# B&R Automation Studio project 8238 (part 20)

#### _actReqScheduleDFII.st
```iecst
(********************************************************************
 * COPYRIGHT -- Herbert Kannegiesser GmbH
 ********************************************************************
 * Program: hlDFII
 * File: _actReqScheduleDFII.st
 * Author: hunholz
 * Created: June 20, 2012
 ********************************************************************
 * Implementation of program hlDFII
 ********************************************************************)

(* Process Requests for DFII *)
ACTION _actReqScheduleDFII:

	// Der Scheduler wird nur ausgeführt, wenn kein SQL-Commando bearbeitet wird

	IF _eCmdDFIIStep = eCMD_SQLREQ_IDLE THEN

		CASE _wScheduleStep OF

			_HLDFII_SCHEDSTEP_GETTIME:

				// Uhrzeit holen
				IF _bEventGetTime = _HLDFII_REQ_START THEN
					// Auftrag starten
					_eCmdDFIIStep := eCMD_SQLREQ_WRITE_GETTIME;
					_bEventGetTime := _HLDFII_REQ_RUN;
				END_IF

			_HLDFII_SCHEDSTEP_REGMACHINE:

				// Maschine registrieren
				IF _bEventRegMach = _HLDFII_REQ_START AND brwcscmp(ADR(IFmnParam.Out.utfMachineNumber),ADR(MNPARAM_INVALID_MACHINENO)) <> 0 THEN
					// Auftrag starten
					_eCmdDFIIStep := eCMD_SQLREQ_WRITE_REGMACH;
					_bEventRegMach := _HLDFII_REQ_RUN;
				END_IF

			_HLDFII_SCHEDSTEP_PROGBYCAT:

				// Programmnummer anhand der Kategorie ermitteln
				IF _xWaitReqProgByCatIsZero THEN

					IF IFhlDFII.In.ReqProgByCat.wRequest = 0 THEN

						_xWaitReqProgByCatIsZero := FALSE;
						IFhlDFII.Out.RespProgByCat.wResponse := 0;

					END_IF

				ELSE

					// Prüfen ob eine Programmnummer gelesen werden soll
					IF IFhlDFII.In.ReqProgByCat.wRequest = 1 OR IFhlDFII.In.ReqProgByCat.wRequest = 2 THEN

						IF IFhlDFII.Out.xConnected THEN

							_xWaitReqProgByCatIsZero := TRUE;
							// Auftrag starten
							_eCmdDFIIStep := eCMD_SQLREQ_GET_PROG_BY_CAT;
							IFhlDFII.Out.RespProgByCat.wResponse := ERR_FUB_BUSY;

						ELSE

							_xWaitReqProgByCatIsZero := TRUE;
							IFhlDFII.Out.RespProgByCat.wResponse := HLDFII_STAT_NO_CONNECTION;

						END_IF

					END_IF

				END_IF

			_HLDFII_SCHEDSTEP_MSGEVENT:

				// Meldungden senden
				IF _xWaitReqMsgEvtIsZero THEN

					IF IFhlDFII.In.ReqMsgEvt.wRequest = 0 THEN
						_xWaitReqMsgEvtIsZero := FALSE;
						IFhlDFII.Out.RespMsgEvt.wResponse := 0;
					END_IF

				ELSE

					IF IFhlDFII.Out.xConnected THEN

						// Prüfen ob Meldungsevents geschrieben werden sollen
						IF IFhlDFII.In.ReqMsgEvt.wRequest = 1 THEN

							_xWaitReqMsgEvtIsZero := TRUE;

							IF IFhlDFII.In.ReqMsgEvt.bCntLines > 0 THEN
								_eCmdDFIIStep := eCMD_SQLREQ_WRITE_MSG;
								IFhlDFII.Out.RespMsgEvt.wResponse := ERR_FUB_BUSY;
							ELSE
								IFhlDFII.Out.RespMsgEvt.wResponse := IFhlDFII.In.ReqMsgEvt.wRequest;
							END_IF

						END_IF

					ELSE

						_xWaitReqMsgEvtIsZero := TRUE;
						IFhlDFII.Out.RespMsgEvt.wResponse := HLDFII_STAT_NO_CONNECTION;

					END_IF

				END_IF

			_HLDFII_SCHEDSTEP_CNTBATCH:

				// Postendaten senden
				IF _xWaitReqCntBatchIsZero THEN

					IF IFhlDFII.In.ReqCntBatchEvt.wRequest = 0 THEN

						_xWaitReqCntBatchIsZero := FALSE;
						IFhlDFII.Out.RespCntBatchEvt.wResponse := 0;

					END_IF

				ELSE

					IF IFhlDFII.Out.xConnected THEN

						// Prüfen ob Zähler-Posten-Events geschrieben werden sollen
						IF IFhlDFII.In.ReqCntBatchEvt.wRequest = 1 THEN

							_xWaitReqCntBatchIsZero := TRUE;

							IF IFhlDFII.In.ReqCntBatchEvt.bCntLines > 0 THEN
								_eCmdDFIIStep := eCMD_SQLREQ_WRITE_CNTBATCHEVT;
								IFhlDFII.Out.RespCntBatchEvt.wResponse := ERR_FUB_BUSY;
							ELSE
								IFhlDFII.Out.RespCntBatchEvt.wResponse  := IFhlDFII.In.ReqCntBatchEvt.wRequest;
							END_IF
						END_IF

					ELSE

						_xWaitReqCntBatchIsZero := TRUE;
						IFhlDFII.Out.RespCntBatchEvt.wResponse := HLDFII_STAT_NO_CONNECTION;

					END_IF

				END_IF

			// Zähler senden
			_HLDFII_SCHEDSTEP_CNTCNT:

				IF _xWaitReqCntCntIsZero THEN

					IF IFhlDFII.In.ReqCntCntEvt.wRequest = 0 THEN

						_xWaitReqCntCntIsZero := FALSE;
						IFhlDFII.Out.RespCntCntEvt.wResponse := 0;

					END_IF

				ELSE

					IF IFhlDFII.Out.xConnected THEN

						// Prüfen ob Zähler-Zähler-Events geschrieben werden sollen
						IF IFhlDFII.In.ReqCntCntEvt.wRequest = 1 THEN

							_xWaitReqCntCntIsZero := TRUE;

							IF IFhlDFII.In.ReqCntCntEvt.bCntLines > 0 THEN
								_eCmdDFIIStep := eCMD_SQLREQ_WRITE_CNTCNTEVT;
								IFhlDFII.Out.RespCntCntEvt.wResponse := ERR_FUB_BUSY;
							ELSE
								IFhlDFII.Out.RespCntCntEvt.wResponse  := IFhlDFII.In.ReqCntCntEvt.wRequest;
							END_IF
						END_IF

					ELSE

						_xWaitReqCntCntIsZero := TRUE;
						IFhlDFII.Out.RespCntCntEvt.wResponse := HLDFII_STAT_NO_CONNECTION;

					END_IF

				END_IF

			// Zeiten senden
			_HLDFII_SCHEDSTEP_CNTTIME:

				IF _xWaitReqCntTimIsZero THEN

					IF IFhlDFII.In.ReqCntTimEvt.wRequest = 0 THEN

						_xWaitReqCntTimIsZero := FALSE;
						IFhlDFII.Out.RespCntTimEvt.wResponse := 0;

					END_IF

				ELSE

					IF IFhlDFII.Out.xConnected THEN

						// Prüfen ob Zähler-Zeit-Events geschrieben werden sollen
						IF IFhlDFII.In.ReqCntTimEvt.wRequest = 1 THEN

							_xWaitReqCntTimIsZero := TRUE;

							IF IFhlDFII.In.ReqCntTimEvt.bCntLines > 0 THEN
								_eCmdDFIIStep := eCMD_SQLREQ_WRITE_CNTTIMEVT;
								IFhlDFII.Out.RespCntTimEvt.wResponse := ERR_FUB_BUSY;
							ELSE
								IFhlDFII.Out.RespCntTimEvt.wResponse  := IFhlDFII.In.ReqCntTimEvt.wRequest;
							END_IF
						END_IF

					ELSE

						_xWaitReqCntTimIsZero := TRUE;
						IFhlDFII.Out.RespCntTimEvt.wResponse := HLDFII_STAT_NO_CONNECTION;

					END_IF

				END_IF

			// Dosierungen senden
			_HLDFII_SCHEDSTEP_CNTDOS:

				IF _xWaitReqCntDosIsZero THEN

					IF IFhlDFII.In.ReqCntDosEvt.wRequest = 0 THEN

						_xWaitReqCntDosIsZero := FALSE;
						IFhlDFII.Out.RespCntDosEvt.wResponse := 0;

					END_IF

				ELSE

					IF IFhlDFII.Out.xConnected THEN

						// Prüfen ob Zähler-Dosier-Events geschrieben werden sollen
						IF IFhlDFII.In.ReqCntDosEvt.wRequest = 1 THEN

							_xWaitReqCntDosIsZero := TRUE;

							IF IFhlDFII.In.ReqCntDosEvt.bCntLines > 0 THEN
								_eCmdDFIIStep := eCMD_SQLREQ_WRITE_CNTDOSEVT;
								IFhlDFII.Out.RespCntDosEvt.wResponse := ERR_FUB_BUSY;
							ELSE
								IFhlDFII.Out.RespCntDosEvt.wResponse  := IFhlDFII.In.ReqCntDosEvt.wRequest;
							END_IF

						END_IF

					ELSE

						_xWaitReqCntDosIsZero := TRUE;
						IFhlDFII.Out.RespCntDosEvt.wResponse := HLDFII_STAT_NO_CONNECTION;

					END_IF

				END_IF

		END_CASE

	END_IF

END_ACTION
```

#### _actProcCmdTrack.st
```iecst
(********************************************************************
 * COPYRIGHT -- Herbert Kannegiesser GmbH
 ********************************************************************
 * Program: hlDFII
 * File: _actProcCmdTrack.st
 * Author: hunholz
 * Created: June 20, 2012
 ********************************************************************
 * Implementation of program hlDFII
 ********************************************************************)

(* Process Commands for DFII *)
ACTION _actProcCmdTrack:

	_TONRefreshTrack(IN := NOT _TONRefreshTrack.Q, PT := T#1s);

	CASE _eCmdTrackStep OF

		//*****************************************************
		// Im Idle Zustand werden laufend die Auftrage gescannt
		//*****************************************************
		eCMD_SQLREQ_IDLE:

			// Zuerst wird die Zeit vom Server geholt
			IF _bEventGetTrackTime <> _HLDFII_REQ_FINISHED THEN

				_wScheduleTrackStep := _HLDFII_SCHEDSTEP_T_GETTIME;

				// Dann wird zyklisch geschaut, ob Anforderungen anliegen
			ELSE

				IF _TONRefreshTrack.Q THEN

					_wScheduleTrackStepHelp := (_wScheduleTrackStepHelp + 1) MOD (_HLDFII_SCHEDSTEP_T_MAX);

					_wScheduleTrackStep := _wScheduleTrackStepHelp + 1;

				END_IF

			END_IF

		//*****************************************************
		// Uhrzeit vom DB-Server holen
		//*****************************************************
		eCMD_SQLREQ_WRITE_GETTIME:

			IF _eTrackStep = eSQLREQ_STEP_WAITFORCOMMAND THEN

				_eTrackStep := eSQLREQ_STEP_GETTIME;
				_eCmdTrackStep := eCMD_SQLREQ_WRITE_GETTIME_w;

			ELSIF _eTrackStep = eSQLREQ_STEP_ERROR THEN

				_bEventGetTrackTime := _HLDFII_REQ_FAULT;
				_eCmdTrackStep := eCMD_SQLREQ_IDLE;

			END_IF

		eCMD_SQLREQ_WRITE_GETTIME_w:

			IF _eTrackStep = eSQLREQ_STEP_WAITFORCOMMAND THEN

				_bEventGetTrackTime := _HLDFII_REQ_FINISHED;
				_eCmdTrackStep := eCMD_SQLREQ_IDLE;

			ELSIF _eTrackStep = eSQLREQ_STEP_ERROR THEN

				_bEventGetTrackTime := _HLDFII_REQ_FAULT;
				_eCmdTrackStep := eCMD_SQLREQ_IDLE;

			END_IF

		//***************************************
		// Batchdaten in Location-Table eintragen
		//***************************************
		eCMD_SQLREQ_WRITE_UPDLOC:

			IF _eTrackStep = eSQLREQ_STEP_WAITFORCOMMAND THEN

				_wIdxWriteUpdateLocation := 1;
				_eTrackStep := eSQLREQ_STEP_WRUPDLOC;
				_eCmdTrackStep := eCMD_SQLREQ_WRITE_UPDLOC_w;

			ELSIF _eTrackStep = eSQLREQ_STEP_ERROR THEN

				_xUpdateLocationFinished := TRUE;
				_eCmdTrackStep := eCMD_SQLREQ_IDLE;

			END_IF

		eCMD_SQLREQ_WRITE_UPDLOC_w:

			IF _eTrackStep = eSQLREQ_STEP_WAITFORCOMMAND THEN

				_xUpdateLocationFinished := TRUE;
				_eCmdTrackStep := eCMD_SQLREQ_IDLE;

			ELSIF _eTrackStep = eSQLREQ_STEP_ERROR THEN

				_xUpdateLocationFinished := TRUE;
				_eCmdTrackStep := eCMD_SQLREQ_IDLE;

			END_IF

		//***************************************
		// Maschinenstatus eintragen
		//***************************************
		eCMD_SQLREQ_WRITE_UPDSTATE:

			IF _eTrackStep = eSQLREQ_STEP_WAITFORCOMMAND THEN

				_wIdxWriteUpdateStatus := 1;
				_eTrackStep := eSQLREQ_STEP_WRUPDSTATE;
				_eCmdTrackStep := eCMD_SQLREQ_WRITE_UPDSTATE_w;

			ELSIF _eTrackStep = eSQLREQ_STEP_ERROR THEN

				_xUpdateStatusFinished := TRUE;
				_eCmdTrackStep := eCMD_SQLREQ_IDLE;

			END_IF

		eCMD_SQLREQ_WRITE_UPDSTATE_w:

			IF _eTrackStep = eSQLREQ_STEP_WAITFORCOMMAND THEN

				_xUpdateStatusFinished := TRUE;
				_eCmdTrackStep := eCMD_SQLREQ_IDLE;

			ELSIF _eTrackStep = eSQLREQ_STEP_ERROR THEN

				_xUpdateStatusFinished := TRUE;
				_eCmdTrackStep := eCMD_SQLREQ_IDLE;

			END_IF

	END_CASE

END_ACTION
```

#### _actProcCmdDFII.st
```iecst
(********************************************************************
 * COPYRIGHT -- Herbert Kannegiesser GmbH
 ********************************************************************
 * Program: hlDFII
 * File: _actProcCmdDFII.st
 * Author: hunholz
 * Created: June 20, 2012
 ********************************************************************
 * Implementation of program hlDFII
 ********************************************************************)

(* Process Commands for DFII *)
ACTION _actProcCmdDFII:

	CASE _eCmdDFIIStep OF

		//*****************************************************
		// Im Idle Zustand werden laufend die Auftrage gescannt
		//*****************************************************
		eCMD_SQLREQ_IDLE:

			// Zuerst wird die Zeit vom Server geholt
			IF _bEventGetTime <> _HLDFII_REQ_FINISHED THEN

				_wScheduleStep := _HLDFII_SCHEDSTEP_GETTIME;

				// Die Maschine wird auf jeden Fall registriert
			ELSIF _bEventRegMach <> _HLDFII_REQ_FINISHED THEN

				_wScheduleStep := _HLDFII_SCHEDSTEP_REGMACHINE;

				// Dann wird zyklisch geschaut, ob Anforderungen anliegen
			ELSE

				_wScheduleStepHelp := (_wScheduleStepHelp + 1) MOD (_HLDFII_SCHEDSTEP_MAX-1);

				_wScheduleStep := _wScheduleStepHelp + 2;

			END_IF

		//*****************************************************
		// Auftrag: Programm nach Kategorie auslesen
		//*****************************************************
		eCMD_SQLREQ_GET_PROG_BY_CAT:

			IF _eStep = eSQLREQ_STEP_WAITFORCOMMAND THEN
				IFhlDFII.Out.RespProgByCat.bProgramNo 		:= 0;
				IFhlDFII.Out.RespProgByCat.sProgramName 	:= '';
				IFhlDFII.Out.RespProgByCat.rSoilfactor 		:= 1.0;
				IFhlDFII.Out.RespProgByCat.wLoadrate 		:= 100;
				IFhlDFII.Out.RespProgByCat.wColorIdxFor 	:= 0;
				IFhlDFII.Out.RespProgByCat.wColorIdxBack 	:= 15;
				_eStep := eSQLREQ_STEP_GPBC;
				_eCmdDFIIStep := eCMD_SQLREQ_GET_PROG_BY_CAT_w;

			ELSIF _eStep = eSQLREQ_STEP_ERROR THEN

				IFhlDFII.Out.RespProgByCat.wResponse := HLDFII_MSG_PROGBYCAT_ERR;
				_eCmdDFIIStep := eCMD_SQLREQ_IDLE;

			END_IF

		eCMD_SQLREQ_GET_PROG_BY_CAT_w:

			IF _eStep = eSQLREQ_STEP_WAITFORCOMMAND THEN
				IFhlDFII.Out.RespProgByCat.wResponse := IFhlDFII.In.ReqProgByCat.wRequest;
				_eCmdDFIIStep := eCMD_SQLREQ_IDLE;
			ELSIF _eStep = eSQLREQ_STEP_ERROR THEN
				IFhlDFII.Out.RespProgByCat.wResponse := HLDFII_MSG_PROGBYCAT_ERR;
				_eCmdDFIIStep := eCMD_SQLREQ_IDLE;
			END_IF

		//*****************************************************
		// Meldungen schreiben
		//*****************************************************
		eCMD_SQLREQ_WRITE_MSG:

			IF _eStep = eSQLREQ_STEP_WAITFORCOMMAND THEN
				_bCntWrMsg := 1;
				_eStep := eSQLREQ_STEP_WRMSG;
				_eCmdDFIIStep := eCMD_SQLREQ_WRITE_MSG_w;
			ELSIF _eStep = eSQLREQ_STEP_ERROR THEN
				IFhlDFII.Out.RespMsgEvt.wResponse := HLDFII_MSG_MSGEVT_ERR;
				_eCmdDFIIStep := eCMD_SQLREQ_IDLE;
			END_IF

		eCMD_SQLREQ_WRITE_MSG_w:

			IF _eStep = eSQLREQ_STEP_WAITFORCOMMAND THEN
				IFhlDFII.Out.RespMsgEvt.wResponse := IFhlDFII.In.ReqMsgEvt.wRequest;
				_eCmdDFIIStep := eCMD_SQLREQ_IDLE;
			ELSIF _eStep = eSQLREQ_STEP_ERROR THEN
				IFhlDFII.Out.RespMsgEvt.wResponse := HLDFII_MSG_MSGEVT_ERR;
				_eCmdDFIIStep := eCMD_SQLREQ_IDLE;
			END_IF

		//*****************************************************
		// Posten-Zählevents schreiben
		//*****************************************************
		eCMD_SQLREQ_WRITE_CNTBATCHEVT:

			IF _eStep = eSQLREQ_STEP_WAITFORCOMMAND THEN
				_bCntWrCntBatchEvt := 1;
				_eStep := eSQLREQ_STEP_WRCNTBATCHEVT;
				_eCmdDFIIStep := eCMD_SQLREQ_WRITE_CNTBATCHEVT_w;
			ELSIF _eStep = eSQLREQ_STEP_ERROR THEN
				IFhlDFII.Out.RespCntBatchEvt.wResponse := HLDFII_MSG_CNTBATCHEVT_ERR;
				_eCmdDFIIStep := eCMD_SQLREQ_IDLE;
			END_IF

		eCMD_SQLREQ_WRITE_CNTBATCHEVT_w:

			IF _eStep = eSQLREQ_STEP_WAITFORCOMMAND THEN
				IFhlDFII.Out.RespCntBatchEvt.wResponse := IFhlDFII.In.ReqCntBatchEvt.wRequest;
				_eCmdDFIIStep := eCMD_SQLREQ_IDLE;
			ELSIF _eStep = eSQLREQ_STEP_ERROR THEN
				IFhlDFII.Out.RespCntBatchEvt.wResponse := HLDFII_MSG_CNTBATCHEVT_ERR;
				_eCmdDFIIStep := eCMD_SQLREQ_IDLE;
			END_IF

		//*****************************************************
		// Zählerevents schreiben
		//*****************************************************
		eCMD_SQLREQ_WRITE_CNTCNTEVT:

			IF _eStep = eSQLREQ_STEP_WAITFORCOMMAND THEN
				_bCntWrCntCntEvt := 1;
				_eStep := eSQLREQ_STEP_WRCNTCNTEVT;
				_eCmdDFIIStep := eCMD_SQLREQ_WRITE_CNTCNTEVT_w;
			ELSIF _eStep = eSQLREQ_STEP_ERROR THEN
				IFhlDFII.Out.RespCntCntEvt.wResponse := HLDFII_MSG_CNTCNTEVT_ERR;
				_eCmdDFIIStep := eCMD_SQLREQ_IDLE;
			END_IF

		eCMD_SQLREQ_WRITE_CNTCNTEVT_w:

			IF _eStep = eSQLREQ_STEP_WAITFORCOMMAND THEN
				IFhlDFII.Out.RespCntCntEvt.wResponse := IFhlDFII.In.ReqCntCntEvt.wRequest;
				_eCmdDFIIStep := eCMD_SQLREQ_IDLE;
			ELSIF _eStep = eSQLREQ_STEP_ERROR THEN
				IFhlDFII.Out.RespCntCntEvt.wResponse := HLDFII_MSG_CNTCNTEVT_ERR;
				_eCmdDFIIStep := eCMD_SQLREQ_IDLE;
			END_IF

		//*****************************************************
		// Zeitevents schreiben
		//*****************************************************
		eCMD_SQLREQ_WRITE_CNTTIMEVT:

			IF _eStep = eSQLREQ_STEP_WAITFORCOMMAND THEN
				_bCntWrCntTimeEvt := 1;
				_eStep := eSQLREQ_STEP_WRCNTTIMEVT;
				_eCmdDFIIStep := eCMD_SQLREQ_WRITE_CNTTIMEVT_w;
			ELSIF _eStep = eSQLREQ_STEP_ERROR THEN
				IFhlDFII.Out.RespCntTimEvt.wResponse := HLDFII_MSG_CNTTIMEVT_ERR;
				_eCmdDFIIStep := eCMD_SQLREQ_IDLE;
			END_IF

		eCMD_SQLREQ_WRITE_CNTTIMEVT_w:

			IF _eStep = eSQLREQ_STEP_WAITFORCOMMAND THEN
				IFhlDFII.Out.RespCntTimEvt.wResponse := IFhlDFII.In.ReqCntTimEvt.wRequest;
				_eCmdDFIIStep := eCMD_SQLREQ_IDLE;
			ELSIF _eStep = eSQLREQ_STEP_ERROR THEN
				IFhlDFII.Out.RespCntTimEvt.wResponse := HLDFII_MSG_CNTTIMEVT_ERR;
				_eCmdDFIIStep := eCMD_SQLREQ_IDLE;
			END_IF

		//*****************************************************
		// Dosierevents schreiben
		//*****************************************************
		eCMD_SQLREQ_WRITE_CNTDOSEVT:

			IF _eStep = eSQLREQ_STEP_WAITFORCOMMAND THEN
				_bCntWrCntDoseEvt := 1;
				_eStep := eSQLREQ_STEP_WRCNTDOSEVT;
				_eCmdDFIIStep := eCMD_SQLREQ_WRITE_CNTDOSEVT_W;
			ELSIF _eStep = eSQLREQ_STEP_ERROR THEN
				IFhlDFII.Out.RespCntDosEvt.wResponse := HLDFII_MSG_CNTDOSEVT_ERR;
				_eCmdDFIIStep := eCMD_SQLREQ_IDLE;
			END_IF

		eCMD_SQLREQ_WRITE_CNTDOSEVT_W:

			IF _eStep = eSQLREQ_STEP_WAITFORCOMMAND THEN
				IFhlDFII.Out.RespCntDosEvt.wResponse := IFhlDFII.In.ReqCntDosEvt.wRequest;
				_eCmdDFIIStep := eCMD_SQLREQ_IDLE;
			ELSIF _eStep = eSQLREQ_STEP_ERROR THEN
				IFhlDFII.Out.RespCntDosEvt.wResponse := HLDFII_MSG_CNTDOSEVT_ERR;
				_eCmdDFIIStep := eCMD_SQLREQ_IDLE;
			END_IF

		//*****************************************************
		// Maschine registrieren
		//*****************************************************
		eCMD_SQLREQ_WRITE_REGMACH:

			IF _eStep = eSQLREQ_STEP_WAITFORCOMMAND THEN
				_eStep := eSQLREQ_STEP_REGMACH;
				_eCmdDFIIStep := eCMD_SQLREQ_WRITE_REGMACH_w;
			ELSIF _eStep = eSQLREQ_STEP_ERROR THEN
				_bEventRegMach := 255;
				_eCmdDFIIStep := eCMD_SQLREQ_IDLE;
			END_IF

		eCMD_SQLREQ_WRITE_REGMACH_w:

			IF _eStep = eSQLREQ_STEP_WAITFORCOMMAND THEN
				_bEventRegMach := 3;
				_eCmdDFIIStep := eCMD_SQLREQ_IDLE;
			ELSIF _eStep = eSQLREQ_STEP_ERROR THEN
				_bEventRegMach := 255;
				_eCmdDFIIStep := eCMD_SQLREQ_IDLE;
			END_IF

		//*****************************************************
		// Uhrzeit vom DB-Server holen
		//*****************************************************
		eCMD_SQLREQ_WRITE_GETTIME:

			IF _eStep = eSQLREQ_STEP_WAITFORCOMMAND THEN
				_eStep := eSQLREQ_STEP_GETTIME;
				_eCmdDFIIStep := eCMD_SQLREQ_WRITE_GETTIME_w;
			ELSIF _eStep = eSQLREQ_STEP_ERROR THEN
				_bEventGetTime := 255;
				_eCmdDFIIStep := eCMD_SQLREQ_IDLE;
			END_IF

		eCMD_SQLREQ_WRITE_GETTIME_w:

			IF _eStep = eSQLREQ_STEP_WAITFORCOMMAND THEN
				_bEventGetTime := 3;
				_eCmdDFIIStep := eCMD_SQLREQ_IDLE;
			ELSIF _eStep = eSQLREQ_STEP_ERROR THEN
				_bEventGetTime := 255;
				_eCmdDFIIStep := eCMD_SQLREQ_IDLE;
			END_IF

	END_CASE

END_ACTION
```

#### _actProcSQLTrack.st
```iecst
(********************************************************************
 * COPYRIGHT -- Herbert Kannegiesser GmbH
 ********************************************************************
 * Program: hlDFII
 * File: _actProcSQLTrack.st
 * Author: hunholz
 * Created: June 20, 2012
 ********************************************************************
 * Implementation of program hlDFII
 ********************************************************************)

(* Process SQL-Queries *)
ACTION _actProcSQLTrack:

	CASE _eTrackStep OF

		eSQLREQ_STEP_STOP:

		eSQLREQ_STEP_WAITFORCOMMAND:

		(* Verbinde Datenbank *)
		eSQLREQ_STEP_CONNECT:

			_Track_Connect.enable := TRUE;
			_Track_Connect.databaseSystem := DB_SYSTEM_MS_SQL;
			_Track_Connect.pUserName := ADR('mas');
			_Track_Connect.pPassword := ADR('1234');
			_Track_Connect.pServerName := ADR(_CreateConnStringTracking.ConnString);
			_Track_Connect.pDatabaseName := ADR(hlDFIIPar.Mac.TrackConn.sDBname);

			_eTrackStep := eSQLREQ_STEP_CONNECT_r;

		(* Warte bis mit Datenbank verbunden *)
		eSQLREQ_STEP_CONNECT_r:

			_Track_Connect();

			IF _Track_Connect.status = ERR_OK THEN

				// Verbindung Erfolgreich

				IF _Track_Connect.connectionIdent = 0 THEN

					// Wenn Verbindung nicht möglich, immer erst wieder Zeit holen
					_bEventGetTrackTime := _HLDFII_REQ_START;
					IFhlDFII.Out.xTrackConnected := FALSE;

					// Fehler ist Clientseitig
					_sLogEntryT := 'Client Fault: Connect failed! ';
					_sLogEntryT := CONCAT(_sLogEntryT,_CreateConnStringTracking.ConnString);
					_eTrackStep := eSQLREQ_STEP_LOGRB_ERROR;

				ELSE

					IFhlDFII.Out.xTrackConnected := TRUE;

					_sLogEntryT := WSTRING_TO_STRING(IFmnParam.Out.utfMachineNumber);
					_sLogEntryT := CONCAT(_sLogEntryT, '-hlDFII$tSUCC$tCONNECT_T');
					_InsertRBT(wPtrWrite := _wPtrRBwrite, wPtrRead := _wPtrRBread, wPtrStart := _wPtrRBstart);

					_lConnectionTrackIdent := _Track_Connect.connectionIdent;
					_eTrackStep := eSQLREQ_STEP_WAITFORCOMMAND;
				END_IF

			ELSIF _Track_Connect.status <> ERR_FUB_BUSY THEN

				// Wenn Verbindung nicht möglich, immer erst wieder Zeit holen und Maschine registrieren
				_bEventGetTrackTime := _HLDFII_REQ_START;
				IFhlDFII.Out.xTrackConnected := FALSE;

				// Verbindung fehlerbehaftet
				IF _Track_Connect.connectionIdent <> 0 THEN

					// Fehler ist Serverseitig, Fehlermeldung holen

					_lConnectionTrackIdent := _Track_Connect.connectionIdent;
					_sTrackAction := 'Connect failed:';
					_eTrackStep := eSQLREQ_STEP_GET_ERROR;

				ELSE

					// Keine Verbindung zustande gekommen
					_sLogEntryT := 'Connect failed! ';
					_sLogEntryT := CONCAT(_sLogEntryT,_CreateConnStringTracking.ConnString);

					_eTrackStep := eSQLREQ_STEP_LOGRB_ERROR;

				END_IF

			END_IF

		(* Baue Datenbankverbindung ab *)
		eSQLREQ_STEP_DISCONNECT:

			IF _lConnectionTrackIdent <> 0 THEN
				_Track_Disconnect.enable := TRUE;
				_Track_Disconnect.connectionIdent := _lConnectionTrackIdent;
				_eTrackStep := eSQLREQ_STEP_DISCONNECT_r;
			ELSE
				_eTrackStep := eSQLREQ_STEP_STOP;
			END_IF

		(* Warte bis Verbindung abgebaut ist *)
		eSQLREQ_STEP_DISCONNECT_r:

			_Track_Disconnect();

			IF _Track_Disconnect.status <> ERR_FUB_BUSY THEN

				// Verbindung erfolgreich unterbrochen

				_sLogEntryT := WSTRING_TO_STRING(IFmnParam.Out.utfMachineNumber);
				_sLogEntryT := CONCAT(_sLogEntryT, '-hlDFII$tSUCC$tDISCONNECT_T');
				_InsertRBT(wPtrWrite := _wPtrRBwrite, wPtrRead := _wPtrRBread, wPtrStart := _wPtrRBstart);

				_eTrackStep := eSQLREQ_STEP_STOP;
				_lConnectionTrackIdent := 0;

			END_IF

		// Uhrzeit von DB lesen
		eSQLREQ_STEP_GETTIME:

			_sSQLstringTrack := 'SELECT DATEDIFF(s,$'1970-01-01T00:00:00$',GETDATE())';

			_Track_DBExecute.enable := TRUE;
			_Track_DBExecute.pSqlStatement := ADR(_sSQLstringTrack);
			_Track_DBExecute.connectionIdent := _lConnectionTrackIdent;

			_eTrackStep := eSQLREQ_STEP_GETTIME_r;

		eSQLREQ_STEP_GETTIME_r:

			_Track_DBExecute();

			IF _Track_DBExecute.status = ERR_OK THEN

				_eTrackStep := eSQLREQ_STEP_GETTIME_FETCH;

			ELSIF _Track_DBExecute.status <> ERR_FUB_BUSY THEN

				_sTrackAction := 'Get Time failed:';
				_eTrackStep := eSQLREQ_STEP_GET_ERROR;

			END_IF

		(* Zeile holen *)
		eSQLREQ_STEP_GETTIME_FETCH:

			_Track_DBFetch.enable := TRUE;
			_Track_DBFetch.connectionIdent := _lConnectionTrackIdent;
			_eTrackStep := eSQLREQ_STEP_GETTIME_FETCH_r;

		eSQLREQ_STEP_GETTIME_FETCH_r:

			_Track_DBFetch();

			IF _Track_DBFetch.status = ERR_OK THEN

				_bTrackCol := 1;
				_eTrackStep := eSQLREQ_STEP_GETTIME_GETVAL;

			ELSIF _Track_DBFetch.status <> ERR_FUB_BUSY THEN

				IF _Track_DBFetch.dbError = DB_SQL_NO_DATA THEN

					_eTrackStep := eSQLREQ_STEP_WAITFORCOMMAND;

				ELSE

					_sTrackAction := 'Get Time failed (FETCH):';
					_eTrackStep := eSQLREQ_STEP_GET_ERROR;

				END_IF

			END_IF

		(* Werte holen *)

		eSQLREQ_STEP_GETTIME_GETVAL:

			_Track_GetData.enable := TRUE;
			_Track_GetData.connectionIdent := _lConnectionTrackIdent;
			_Track_GetData.columnIdx := _bTrackCol;

			_diTimeTrack := -1;
			_Track_GetData.pData := ADR(_diTimeTrack);
			_Track_GetData.dataSize := SIZEOF(_diTimeTrack);
			_Track_GetData.dataType := DB_SQL_INTEGER;

			_eTrackStep := eSQLREQ_STEP_GETTIME_GETVAL_r;

		eSQLREQ_STEP_GETTIME_GETVAL_r:

			_Track_GetData();

			IF _Track_GetData.status = ERR_OK THEN

				IF _diTimeTrack > 0 THEN

					_DTSetTime(enable := TRUE, DT1 := DINT_TO_DT(_diTimeTrack));

				END_IF

				_sLogEntryT := WSTRING_TO_STRING(IFmnParam.Out.utfMachineNumber);
				_sLogEntryT := CONCAT(_sLogEntryT, '-hlDFII$tSUCC$tGETTIME_T');
				_InsertRBT(wPtrWrite := _wPtrRBwrite, wPtrRead := _wPtrRBread, wPtrStart := _wPtrRBstart);

				_eTrackStep := eSQLREQ_STEP_WAITFORCOMMAND;

			ELSIF _Track_GetData.status <> ERR_FUB_BUSY THEN
				_sTrackAction := 'Get Time failed (VAL):';
				_eTrackStep := eSQLREQ_STEP_GET_ERROR;
			END_IF

		eSQLREQ_STEP_WRUPDLOC:

			IF _wIdxWriteUpdateLocation > HLDFII_MAXIDX_REQ_UPDATEBATCH THEN

				_eTrackStep := eSQLREQ_STEP_WAITFORCOMMAND;

			ELSIF _ReqUpdBatch[_wIdxWriteUpdateLocation].wLocation > 0 THEN

				_sSQLstringTrack := 'EXEC [BatchManagement].[uspBatchUpdate] ';
				_sSQLstringTrack := CONCAT(_sSQLstringTrack,'@BatchNumber = ');

				_GetBatchno(usintarray := _ReqUpdBatch[_wIdxWriteUpdateLocation].bBatchNo);
				_lBatchNo := kgBatchNoToUDINT(_GetBatchno.GUID);
				_sTrackValue := UDINT_TO_STRING(_lBatchNo);

				_sSQLstringTrack := CONCAT(_sSQLstringTrack, _sTrackValue);

				_sSQLstringTrack := CONCAT(_sSQLstringTrack,', @MachID = ');
				IF _ReqUpdBatch[_wIdxWriteUpdateLocation].lMachineNo > 0 THEN
					_sTrackValue := UDINT_TO_STRING(_ReqUpdBatch[_wIdxWriteUpdateLocation].lMachineNo);
					_sSQLstringTrack := CONCAT(_sSQLstringTrack, _sTrackValue);
				ELSE
					_sTrackMachineNo := WSTRING_TO_STRING(IFmnParam.Out.utfMachineNumber);
					_sSQLstringTrack := CONCAT(_sSQLstringTrack, _sTrackMachineNo);
				END_IF

				_sSQLstringTrack := CONCAT(_sSQLstringTrack,', @LocationNumber = ');
				_sTrackValue := UDINT_TO_STRING(_ReqUpdBatch[_wIdxWriteUpdateLocation].wLocation);
				_sSQLstringTrack := CONCAT(_sSQLstringTrack, _sTrackValue);

				_sSQLstringTrack := CONCAT(_sSQLstringTrack,', @ElementIndex = ');
				_sTrackValue := UDINT_TO_STRING(_ReqUpdBatch[_wIdxWriteUpdateLocation].wElement);
				_sSQLstringTrack := CONCAT(_sSQLstringTrack, _sTrackValue);

				_sSQLstringTrack := CONCAT(_sSQLstringTrack,', @TimeStamp = $'');
				_mnParam_datetimetoa(dtTimestamp := _ReqUpdBatch[_wIdxWriteUpdateLocation].dtTimeStamp);
				_sSQLstringTrack := CONCAT(_sSQLstringTrack, _mnParam_datetimetoa.sDateTime);
				_sSQLstringTrack := CONCAT(_sSQLstringTrack,'$'');

				_Track_DBExecute.enable := TRUE;
				_Track_DBExecute.pSqlStatement := ADR(_sSQLstringTrack);
				_Track_DBExecute.connectionIdent := _lConnectionTrackIdent;

				_eTrackStep := eSQLREQ_STEP_WRUPDLOC_r;

			ELSE

				_wIdxWriteUpdateLocation := _wIdxWriteUpdateLocation + 1;

			END_IF

		eSQLREQ_STEP_WRUPDLOC_r:

			_Track_DBExecute();

			IF _Track_DBExecute.status = ERR_OK  OR _Track_DBExecute.dbError = DB_SQL_NO_DATA THEN

				_dtTimeStampUpdBatch[_wIdxWriteUpdateLocation] := _ReqUpdBatch[_wIdxWriteUpdateLocation].dtTimeStamp;

				_wIdxWriteUpdateLocation := _wIdxWriteUpdateLocation + 1;
				_eTrackStep := eSQLREQ_STEP_WRUPDLOC;

			ELSIF _Track_DBExecute.status <> ERR_FUB_BUSY THEN

				_dtTimeStampUpdBatch[_wIdxWriteUpdateLocation] := _ReqUpdBatch[_wIdxWriteUpdateLocation].dtTimeStamp;

				_sTrackAction := 'Write Update Location failed:';
				_eTrackStep := eSQLREQ_STEP_GET_ERROR;

			END_IF

		eSQLREQ_STEP_WRUPDSTATE:

			IF _wIdxWriteUpdateStatus > HLDFII_MAXIDX_REQ_UPDATESTATUS THEN

				_eTrackStep := eSQLREQ_STEP_WAITFORCOMMAND;

			ELSIF _ReqUpdStatus[_wIdxWriteUpdateStatus].xEnable AND (
				_ReqUpdStatus[_wIdxWriteUpdateStatus].wStatusX <> _wStatusX[_wIdxWriteUpdateStatus]
				OR _ReqUpdStatus[_wIdxWriteUpdateStatus].wSubState <> _wSubState[_wIdxWriteUpdateStatus]
				OR brsstrcmp(ADR(_ReqUpdStatus[_wIdxWriteUpdateStatus]),ADR(_sSubStates[_wIdxWriteUpdateStatus])) <> 0)THEN

				_sSQLstringTrack := 'EXEC [BatchManagement].[uspMachineStateUpdate] ';

				_sSQLstringTrack := CONCAT(_sSQLstringTrack,' @MachID = ');
				IF _ReqUpdStatus[_wIdxWriteUpdateStatus].lMachineNo > 0 THEN
					_sTrackValue := UDINT_TO_STRING(_ReqUpdStatus[_wIdxWriteUpdateStatus].lMachineNo);
					_sSQLstringTrack := CONCAT(_sSQLstringTrack, _sTrackValue);
				ELSE
					_sTrackMachineNo := WSTRING_TO_STRING(IFmnParam.Out.utfMachineNumber);
					_sSQLstringTrack := CONCAT(_sSQLstringTrack, _sTrackMachineNo);
				END_IF

				_sSQLstringTrack := CONCAT(_sSQLstringTrack,', @MachineState = ');
				_sTrackValue := UINT_TO_STRING(_ReqUpdStatus[_wIdxWriteUpdateStatus].wStatusX AND 16#FF);
				_sSQLstringTrack := CONCAT(_sSQLstringTrack, _sTrackValue);

				_sSQLstringTrack := CONCAT(_sSQLstringTrack,', @MachineStateDesc = N$'');
				IF _ReqUpdStatus[_wIdxWriteUpdateStatus].wStatusX.8 AND NOT _ReqUpdStatus[_wIdxWriteUpdateStatus].wStatusX.9 THEN

					_sSQLstringTrack := CONCAT(_sSQLstringTrack, 'PAUSED');

					CASE _ReqUpdStatus[_wIdxWriteUpdateStatus].wSubState OF

						MNCNT_TIMERSUBSTATE_OFF:

							_sSubState := 'OFF';

						MNCNT_TIMERSUBSTATE_STOP:

							_sSubState := 'STOP';

						MNCNT_TIMERSUBSTATE_INTFAULT:

							_sSubState := 'INTFAULT';

						MNCNT_TIMERSUBSTATE_EXTFAULT:

							_sSubState := 'EXTFAULT';

						MNCNT_TIMERSUBSTATE_SAFESTOP:

							_sSubState := 'SAFESTOM';

						MNCNT_TIMERSUBSTATE_EMERGENCYSTP:

							_sSubState := 'EMERGSTOP';

						ELSE

							_sSubState := '';

					END_CASE

				ELSIF NOT _ReqUpdStatus[_wIdxWriteUpdateStatus].wStatusX.8 AND _ReqUpdStatus[_wIdxWriteUpdateStatus].wStatusX.9 THEN
					_sSQLstringTrack := CONCAT(_sSQLstringTrack, 'WAIT');

					CASE _ReqUpdStatus[_wIdxWriteUpdateStatus].wSubState OF

						MNCNT_TIMERSUBSTATE_LOADING:

							_sSubState := 'LOADING';

						MNCNT_TIMERSUBSTATE_UNLOADING:

							_sSubState := 'UNLOADING';

						MNCNT_TIMERSUBSTATE_DOSING:

							_sSubState := 'DOSING';

						MNCNT_TIMERSUBSTATE_WATERLEVEL:

							_sSubState := 'WATERLEVEL';

						MNCNT_TIMERSUBSTATE_TEMPERATURE:

							_sSubState := 'TEMP';

						MNCNT_TIMERSUBSTATE_DISINFECTION:

							_sSubState := 'DISINFECTION';

						MNCNT_TIMERSUBSTATE_AIRPRESSURE:

							_sSubState := 'AIRPRESS';

						ELSE

							_sSubState := '';

					END_CASE

				ELSE
					_sSQLstringTrack := CONCAT(_sSQLstringTrack, 'ACTIVE');

					CASE _ReqUpdStatus[_wIdxWriteUpdateStatus].wSubState OF

						MNCNT_TIMERSUBSTATE_WASHING:

							_sSubState := 'PROCESSING';

						MNCNT_TIMERSUBSTATE_PREPERATION:

							_sSubState := 'PREPERATION';

						MNCNT_TIMERSUBSTATE_TRANSFER:

							_sSubState := 'TRANSFER';

						MNCNT_TIMERSUBSTATE_PREPFORSTOP:

							_sSubState := 'PREPFORSTOP';

						ELSE

							_sSubState := '';

					END_CASE

				END_IF
				_sSQLstringTrack := CONCAT(_sSQLstringTrack,'$'');

				_sSQLstringTrack := CONCAT(_sSQLstringTrack,', @MachineSubState = N$'');

				IF brsstrcmp(ADR(_ReqUpdStatus[_wIdxWriteUpdateStatus].sSubState),ADR('')) <> 0 THEN

					_sSQLstringTrack := CONCAT(_sSQLstringTrack, _ReqUpdStatus[_wIdxWriteUpdateStatus].sSubState);

				ELSE

					_sSQLstringTrack := CONCAT(_sSQLstringTrack, _sSubState);

				END_IF

				_sSQLstringTrack := CONCAT(_sSQLstringTrack,'$'');

				_Track_DBExecute.enable := TRUE;
				_Track_DBExecute.pSqlStatement := ADR(_sSQLstringTrack);
				_Track_DBExecute.connectionIdent := _lConnectionTrackIdent;

				_eTrackStep := eSQLREQ_STEP_WRUPDSTATE_r ;

			ELSE

				_wIdxWriteUpdateStatus := _wIdxWriteUpdateStatus + 1;

			END_IF

		eSQLREQ_STEP_WRUPDSTATE_r:

			_Track_DBExecute();

			IF _Track_DBExecute.status = ERR_OK  OR _Track_DBExecute.dbError = DB_SQL_NO_DATA THEN

				_wStatusX[_wIdxWriteUpdateStatus] := _ReqUpdStatus[_wIdxWriteUpdateStatus].wStatusX;
				_wSubState[_wIdxWriteUpdateStatus] := _ReqUpdStatus[_wIdxWriteUpdateStatus].wSubState;
				_sSubStates[_wIdxWriteUpdateStatus] := _ReqUpdStatus[_wIdxWriteUpdateStatus].sSubState;

				_wIdxWriteUpdateStatus := _wIdxWriteUpdateStatus + 1;
				_eTrackStep := eSQLREQ_STEP_WRUPDSTATE;

			ELSIF _Track_DBExecute.status <> ERR_FUB_BUSY THEN

				_wStatusX[_wIdxWriteUpdateStatus] := _ReqUpdStatus[_wIdxWriteUpdateStatus].wStatusX;

				_sTrackAction := 'Write Update Status failed:';
				_eTrackStep := eSQLREQ_STEP_GET_ERROR;

			END_IF

		(* Lese Fehler aus *)
		eSQLREQ_STEP_GET_ERROR:

			IF _lConnectionTrackIdent = 0 THEN
				IFhlDFII.Out.sStatusTracking := 'Connect failed !';
				_eTrackStep := eSQLREQ_STEP_ERROR;
			ELSE
				_Track_DBErrMsg.enable := TRUE;
				_Track_DBErrMsg.connectionIdent := _lConnectionTrackIdent;
				_Track_DBErrMsg.pErrorMessage := ADR(IFhlDFII.Out.sStatusTracking);
				_Track_DBErrMsg.errorMessageSize := SIZEOF(IFhlDFII.Out.sStatusTracking);
				_eTrackStep := eSQLREQ_STEP_GET_ERROR_r;
			END_IF

		(* Warte bis Fehler ausgelesen *)
		eSQLREQ_STEP_GET_ERROR_r:

			_Track_DBErrMsg();

			IF _Track_DBErrMsg.status = ERR_OK THEN

				_sLogEntryT := WSTRING_TO_STRING(IFmnParam.Out.utfMachineNumber);
				_sLogEntryT := CONCAT(_sLogEntryT, '-hlDFII$tWARN$t');
				_sLogEntryT := CONCAT(_sLogEntryT, _sTrackAction);
				_sLogEntryT := CONCAT(_sLogEntryT, IFhlDFII.Out.sStatusTracking);

				_eTrackStep := eSQLREQ_STEP_LOGRB_ERROR;

			ELSIF _Track_DBErrMsg.status <> ERR_FUB_BUSY THEN

				IFhlDFII.Out.sStatusTracking := ' DBErrMsg.status = ';
				_sTrackValue := UINT_TO_STRING(_Track_DBErrMsg.status);
				IFhlDFII.Out.sStatusTracking := CONCAT(IFhlDFII.Out.sStatusTracking, _sTrackValue);

				_sLogEntryT := WSTRING_TO_STRING(IFmnParam.Out.utfMachineNumber);
				_sLogEntryT := CONCAT(_sLogEntryT, '-hlDFII$tWARN$t');
				_sLogEntryT := CONCAT(_sLogEntryT, _sTrackAction);
				_sLogEntryT := CONCAT(_sLogEntryT, IFhlDFII.Out.sStatusTracking);

				_eTrackStep := eSQLREQ_STEP_LOGRB_ERROR;

			END_IF

		eSQLREQ_STEP_LOGRB_ERROR:

			_InsertRBT(wPtrWrite := _wPtrRBwrite, wPtrRead := _wPtrRBread, wPtrStart := _wPtrRBstart);
			_eTrackStep := eSQLREQ_STEP_LOG_ERROR;

		eSQLREQ_STEP_LOG_ERROR:

			_kgArLogWriteTrack.logLevel 	:= arlogLEVEL_WARNING;
			_kgArLogWriteTrack.text		:= LEFT(_sLogEntryT, 127);
			_kgArLogWriteTrack();

			IF _kgArLogWriteTrack.status <> ERR_FUB_BUSY THEN
				brsmemset(ADR(_sLogEntryT), 0, SIZEOF(_sLogEntryT));
				_eTrackStep := eSQLREQ_STEP_LOG_ERROR1;
			END_IF

		eSQLREQ_STEP_LOG_ERROR1:

			_kgArLogWriteTrack.logLevel 	:= arlogLEVEL_WARNING;
			_kgArLogWriteTrack.text		:= LEFT(_sSQLstringTrack, 127);
			_kgArLogWriteTrack();

			IF _kgArLogWriteTrack.status <> ERR_FUB_BUSY THEN
				_eTrackStep := eSQLREQ_STEP_ERROR;
			END_IF

		(* Fehlerschritt *)
		eSQLREQ_STEP_ERROR:

	END_CASE

END_ACTION
```

#### _actProcSQLDFII.st
```iecst
(********************************************************************
 * COPYRIGHT -- Herbert Kannegiesser GmbH
 ********************************************************************
 * Program: hlDFII
 * File: _actProcSQLDFII.st
 * Author: hunholz
 * Created: June 20, 2012
 ********************************************************************
 * Implementation of program hlDFII
 ********************************************************************)

(* Process SQL-Queries *)
ACTION _actProcSQLDFII:

	CASE _eStep OF

		eSQLREQ_STEP_STOP:

		eSQLREQ_STEP_WAITFORCOMMAND:

		(* Verbinde Datenbank *)
		eSQLREQ_STEP_CONNECT:

			_DFII_Connect.enable := TRUE;
			_DFII_Connect.databaseSystem := DB_SYSTEM_MS_SQL;
			_DFII_Connect.pUserName := ADR('plc');
			_DFII_Connect.pPassword := ADR('plc');
			_DFII_Connect.pServerName := ADR(_CreateConnStringDFII.ConnString);
			_DFII_Connect.pDatabaseName := ADR(hlDFIIPar.Mac.DFIIConn.sDBname);
			_eStep := eSQLREQ_STEP_CONNECT_r;

		(* Warte bis mit Datenbank verbunden *)
		eSQLREQ_STEP_CONNECT_r:

			_DFII_Connect();

			IF _DFII_Connect.status = ERR_OK THEN

				// Verbindung Erfolgreich

				IF _DFII_Connect.connectionIdent = 0 THEN

					// Wenn Verbindung nicht möglich, immer erst wieder Zeit holen und Maschine registrieren
					_bEventRegMach := 1;
					_bEventGetTime := 1;
					IFhlDFII.Out.xConnected := FALSE;

					// Fehler ist Clientseitig
					_sLogEntryI := 'Client Fault: Connect failed! ';
					_sLogEntryI := CONCAT(_sLogEntryI,_CreateConnStringDFII.ConnString);
					_eStep := eSQLREQ_STEP_LOGRB_ERROR;

				ELSE

					IFhlDFII.Out.xConnected := TRUE;

					_sLogEntryI := WSTRING_TO_STRING(IFmnParam.Out.utfMachineNumber);
					_sLogEntryI := CONCAT(_sLogEntryI, '-hlDFII$tSUCC$tCONNECT');
					_InsertRB(wPtrWrite := _wPtrRBwrite, wPtrRead := _wPtrRBread, wPtrStart := _wPtrRBstart);

					_lConnectionIdent := _DFII_Connect.connectionIdent;
					_eStep := eSQLREQ_STEP_WAITFORCOMMAND;
				END_IF

			ELSIF _DFII_Connect.status <> ERR_FUB_BUSY THEN

				// Wenn Verbindung nicht möglich, immer erst wieder Zeit holen und Maschine registrieren
				_bEventRegMach := 1;
				_bEventGetTime := 1;
				IFhlDFII.Out.xConnected := FALSE;

				// Verbindung fehlerbehaftet
				IF _DFII_Connect.connectionIdent <> 0 THEN

					// Fehler ist Serverseitig, Fehlermeldung holen

					_lConnectionIdent := _DFII_Connect.connectionIdent;
					_sAction := 'Connect failed:';
					_eStep := eSQLREQ_STEP_GET_ERROR;

				ELSE

					// Keine Verbindung zustande gekommen
					_sLogEntryI := 'Connect failed! ';
					_sLogEntryI := CONCAT(_sLogEntryI,_CreateConnStringDFII.ConnString);

					_eStep := eSQLREQ_STEP_LOGRB_ERROR;

				END_IF

			END_IF

		(* Baue Datenbankverbindung ab *)
		eSQLREQ_STEP_DISCONNECT:

			IF _lConnectionIdent <> 0 THEN
				_DFII_Disconnect.enable := TRUE;
				_DFII_Disconnect.connectionIdent := _lConnectionIdent;
				_eStep := eSQLREQ_STEP_DISCONNECT_r;
			ELSE
				_eStep := eSQLREQ_STEP_STOP;
			END_IF

		(* Warte bis Verbindung abgebaut ist *)
		eSQLREQ_STEP_DISCONNECT_r:

			_DFII_Disconnect();

			IF _DFII_Disconnect.status <> ERR_FUB_BUSY THEN

				// Verbindung erfolgreich unterbrochen

				_sLogEntryI := WSTRING_TO_STRING(IFmnParam.Out.utfMachineNumber);
				_sLogEntryI := CONCAT(_sLogEntryI, '-hlDFII$tSUCC$tDISCONNECT');
				_InsertRB(wPtrWrite := _wPtrRBwrite, wPtrRead := _wPtrRBread, wPtrStart := _wPtrRBstart);

				_eStep := eSQLREQ_STEP_STOP;
				_lConnectionIdent := 0;

			END_IF

		(* Lese Programmnummer aus Datenbank *)
		eSQLREQ_STEP_GPBC:

			_sCat := IFhlDFII.In.ReqProgByCat.sCategoryNo_In;

			brsstrcpy(ADR(_sSQLstring), ADR('SELECT [ProgramNo], [ProgramName], [CategoryName], [LoadFactor], [SoiledFactor], [fgColorIndex], [bgColorIndex]  FROM [dbo].[vwCatToProg01] WHERE [MachineID] = N$''));
			brsstrcat(ADR(_sSQLstring), ADR(_sMNo));
			IF (IFhlDFII.In.ReqProgByCat.wRequest = 2) THEN
				brsstrcat(ADR(_sSQLstring),ADR('$' AND  LTRIM(RTRIM(CategoryNoAlpha)) =  LTRIM(RTRIM($''));
			ELSE
				brsstrcat(ADR(_sSQLstring),ADR('$' AND [CategoryNo] = '));
			END_IF
			brsstrcat(ADR(_sSQLstring),ADR(_sCat));
			IF (IFhlDFII.In.ReqProgByCat.wRequest = 2) THEN
				brsstrcat(ADR(_sSQLstring),ADR('$'))'));
			END_IF

			_DFII_DBExecute.enable := TRUE;
			_DFII_DBExecute.pSqlStatement := ADR(_sSQLstring);
			_DFII_DBExecute.connectionIdent := _lConnectionIdent;

			_eStep := eSQLREQ_STEP_GPBC_r;

		eSQLREQ_STEP_GPBC_r:

			_DFII_DBExecute();

			IF _DFII_DBExecute.status = ERR_OK THEN

				_eStep := eSQLREQ_STEP_GPBC_FETCH;

			ELSIF _DFII_DBExecute.status <> ERR_FUB_BUSY THEN

				IF _DFII_DBExecute.dbError = DB_SQL_NO_DATA THEN

					_eStep := eSQLREQ_STEP_WAITFORCOMMAND;

				ELSE

					_sAction := 'Get Program failed:';
					_eStep := eSQLREQ_STEP_GET_ERROR;

				END_IF

			END_IF

		(* Zeile holen *)
		eSQLREQ_STEP_GPBC_FETCH:

			_DFII_DBFetch.enable := TRUE;
			_DFII_DBFetch.connectionIdent := _lConnectionIdent;
			_eStep := eSQLREQ_STEP_GPBC_FETCH_r;

		eSQLREQ_STEP_GPBC_FETCH_r:

			_DFII_DBFetch();

			IF _DFII_DBFetch.status = ERR_OK THEN

				_bCol := 1;
				_eStep := eSQLREQ_STEP_GPBC_GETVAL;

			ELSIF _DFII_DBFetch.status <> ERR_FUB_BUSY THEN

				IF _DFII_DBFetch.dbError = DB_SQL_NO_DATA THEN

					_eStep := eSQLREQ_STEP_WAITFORCOMMAND;

				ELSE

					_sAction := 'Get Program failed (FETCH):';
					_eStep := eSQLREQ_STEP_GET_ERROR;

				END_IF

			END_IF

		(* Werte holen *)

		eSQLREQ_STEP_GPBC_GETVAL:

			_DFII_GetData.enable := TRUE;
			_DFII_GetData.connectionIdent := _lConnectionIdent;
			_DFII_GetData.columnIdx := _bCol;

			CASE _bCol OF

				1:	_DFII_GetData.pData := ADR(_iProgNo);
					_DFII_GetData.dataSize := SIZEOF(_iProgNo);
					_DFII_GetData.dataType := DB_SQL_SMALLINT;

				2: 	_DFII_GetData.pData := ADR(IFhlDFII.Out.RespProgByCat.sProgramName);
					_DFII_GetData.dataSize := SIZEOF(IFhlDFII.Out.RespProgByCat.sProgramName);
					_DFII_GetData.dataType := DB_SQL_CHAR;

				3: 	_DFII_GetData.pData := ADR(IFhlDFII.Out.RespProgByCat.sCategoryName);
					_DFII_GetData.dataSize := SIZEOF(IFhlDFII.Out.RespProgByCat.sCategoryName);
					_DFII_GetData.dataType := DB_SQL_CHAR;

				4: 	_DFII_GetData.pData := ADR(_rLoadfactor);
					_DFII_GetData.dataSize := SIZEOF(_rLoadfactor);
					_DFII_GetData.dataType := DB_SQL_REAL;

				5: 	_DFII_GetData.pData := ADR(IFhlDFII.Out.RespProgByCat.rSoilfactor);
					_DFII_GetData.dataSize := SIZEOF(IFhlDFII.Out.RespProgByCat.rSoilfactor);
					_DFII_GetData.dataType := DB_SQL_REAL;

				6: 	_DFII_GetData.pData := ADR(_diColIdxFor);
					_DFII_GetData.dataSize := SIZEOF(_diColIdxFor);
					_DFII_GetData.dataType := DB_SQL_INTEGER;

				7: 	_DFII_GetData.pData := ADR(_diColIdxBack);
					_DFII_GetData.dataSize := SIZEOF(_diColIdxBack);
					_DFII_GetData.dataType := DB_SQL_INTEGER;

			END_CASE

			_eStep := eSQLREQ_STEP_GPBC_GETVAL_r;

		eSQLREQ_STEP_GPBC_GETVAL_r:

			_DFII_GetData();

			IF _DFII_GetData.status = ERR_OK THEN

				_bCol := _bCol + 1;

				IF _bCol <= 7 THEN
					_eStep := eSQLREQ_STEP_GPBC_GETVAL;
				ELSE
					IF _iProgNo >= 0 AND _iProgNo <= 99 THEN

						IFhlDFII.Out.RespProgByCat.bProgramNo := INT_TO_USINT(_iProgNo);
						IFhlDFII.Out.RespProgByCat.wLoadrate := REAL_TO_UINT(_rLoadfactor);
						IFhlDFII.Out.RespProgByCat.wColorIdxFor := DINT_TO_UINT(_diColIdxFor);
						IFhlDFII.Out.RespProgByCat.wColorIdxBack := DINT_TO_UINT(_diColIdxBack);

					ELSE

						IFhlDFII.Out.RespProgByCat.bProgramNo := 0;
						IFhlDFII.Out.RespProgByCat.wLoadrate := 100;
						IFhlDFII.Out.RespProgByCat.wColorIdxFor := 0;
						IFhlDFII.Out.RespProgByCat.wColorIdxBack := 15;

					END_IF

					_sLogEntryI := WSTRING_TO_STRING(IFmnParam.Out.utfMachineNumber);
					_sLogEntryI := CONCAT(_sLogEntryI, '-hlDFII$tSUCC$tGET PROG BY CAT');
					_InsertRB(wPtrWrite := _wPtrRBwrite, wPtrRead := _wPtrRBread, wPtrStart := _wPtrRBstart);

					_eStep := eSQLREQ_STEP_WAITFORCOMMAND;

				END_IF

			ELSIF _DFII_GetData.status <> ERR_FUB_BUSY THEN
				_sAction := 'Get Program failed (VAL):';
				_eStep := eSQLREQ_STEP_GET_ERROR;
			END_IF

		// Meldungen per Prozedur schreiben
		eSQLREQ_STEP_WRMSG:

			IF _bCntWrMsg > IFhlDFII.In.ReqMsgEvt.bCntLines THEN

				_eStep := eSQLREQ_STEP_WAITFORCOMMAND;

			ELSE

				brsstrcpy(ADR(_sSQLstring), ADR('EXEC [dbo].[spInsMsgEvt01]  @MachineID = N$''));
				brsstrcat(ADR(_sSQLstring), ADR(_sMNo));
				brsstrcat(ADR(_sSQLstring), ADR('$''));

				brsstrcat(ADR(_sSQLstring),ADR(', @FunctionID = '));
				brsitoa(IFhlDFII.In.ReqMsgEvt.MsgHistList[_bCntWrMsg].wFunction_ID,ADR(_sFunctionID));
				brsstrcat(ADR(_sSQLstring),ADR(_sFunctionID));

				brsstrcat(ADR(_sSQLstring),ADR(', @MsgNo = '));
				brsitoa(IFhlDFII.In.ReqMsgEvt.MsgHistList[_bCntWrMsg].wMsgNumber,ADR(_sMsgNo));
				brsstrcat(ADR(_sSQLstring),ADR(_sMsgNo));

				brsstrcat(ADR(_sSQLstring),ADR(', @Instance = '));
				brsitoa(IFhlDFII.In.ReqMsgEvt.MsgHistList[_bCntWrMsg].wInstance,ADR(_sInstance));
				brsstrcat(ADR(_sSQLstring),ADR(_sInstance));

				brsstrcat(ADR(_sSQLstring),ADR(', @MsgClass = '));
				brsitoa(IFhlDFII.In.ReqMsgEvt.MsgHistList[_bCntWrMsg].wMsgClass,ADR(_sClass));
				brsstrcat(ADR(_sSQLstring),ADR(_sClass));

				brsstrcat(ADR(_sSQLstring),ADR(', @Event = '));
				brsitoa(IFhlDFII.In.ReqMsgEvt.MsgHistList[_bCntWrMsg].wEvent,ADR(_sEvent));
				brsstrcat(ADR(_sSQLstring),ADR(_sEvent));

				brsstrcat(ADR(_sSQLstring),ADR(', @TimeStamp = '));
				brsitoa(DT_TO_DINT(IFhlDFII.In.ReqMsgEvt.MsgHistList[_bCntWrMsg].TimeStampEvent),ADR(_sTimeStamp));
				brsstrcat(ADR(_sSQLstring),ADR(_sTimeStamp));

				brsstrcat(ADR(_sSQLstring),ADR(', @Time = '));
				brsitoa(IFhlDFII.In.ReqMsgEvt.MsgHistList[_bCntWrMsg].lTime,ADR(_sTime));
				brsstrcat(ADR(_sSQLstring),ADR(_sTime));

				// ##AH20111118
				brsstrcat(ADR(_sSQLstring),ADR(', @Attr1 = $''));
				brsstrcat(ADR(_sSQLstring),ADR(IFhlDFII.In.ReqMsgEvt.MsgHistList[_bCntWrMsg].sAttrTxt));

				brsstrcat(ADR(_sSQLstring),ADR('$', @Attr2 = '));
				brsitoa(IFhlDFII.In.ReqMsgEvt.MsgHistList[_bCntWrMsg].diAttr1,ADR(_sValue));
				brsstrcat(ADR(_sSQLstring),ADR(_sValue));

				brsstrcat(ADR(_sSQLstring),ADR(', @Attr3 = '));
				brsitoa(IFhlDFII.In.ReqMsgEvt.MsgHistList[_bCntWrMsg].diAttr2,ADR(_sValue));
				brsstrcat(ADR(_sSQLstring),ADR(_sValue));

				_DFII_DBExecute.enable := TRUE;
				_DFII_DBExecute.pSqlStatement := ADR(_sSQLstring);
				_DFII_DBExecute.connectionIdent := _lConnectionIdent;

				_eStep := eSQLREQ_STEP_WRMSG_r;

			END_IF

		eSQLREQ_STEP_WRMSG_r:

			_DFII_DBExecute();

			IF _DFII_DBExecute.status = ERR_OK  OR _DFII_DBExecute.dbError = DB_SQL_NO_DATA THEN

				_sLogEntryI := WSTRING_TO_STRING(IFmnParam.Out.utfMachineNumber);
				_sLogEntryI := CONCAT(_sLogEntryI, '-hlDFII$tSUCC$tWRITE MESSAGE');
				_InsertRB(wPtrWrite := _wPtrRBwrite, wPtrRead := _wPtrRBread, wPtrStart := _wPtrRBstart);

				_bCntWrMsg := _bCntWrMsg + 1;
				_eStep := eSQLREQ_STEP_WRMSG;

			ELSIF _DFII_DBExecute.status <> ERR_FUB_BUSY THEN

				_sAction := 'Write Msg failed:';

				_eStep := eSQLREQ_STEP_GET_ERROR;

			END_IF

		// Postendaten schreiben
		eSQLREQ_STEP_WRCNTBATCHEVT:

			IF _bCntWrCntBatchEvt > IFhlDFII.In.ReqCntBatchEvt.bCntLines THEN

				_eStep := eSQLREQ_STEP_WAITFORCOMMAND;

			ELSE

				CASE IFhlDFII.In.ReqCntBatchEvt.CntBatchEvtList[_bCntWrCntBatchEvt].bEvent OF

					MNCNT_BATCHEVENT_LOAD, MNCNT_BATCHEVENT_UNLOAD:

						_sSQLstring := 'EXEC [dbo].[spInsEventStat] ';

						_kgUSINT16toGUID(usintarray := IFhlDFII.In.ReqCntBatchEvt.CntBatchEvtList[_bCntWrCntBatchEvt].Batch.bBatchNo);

						IF IFhlDFII.In.ReqCntBatchEvt.CntBatchEvtList[_bCntWrCntBatchEvt].Batch.bTypeBatchNo = 0 THEN

							brsstrcat(ADR(_sSQLstring), ADR('@BatchID_INT = '));
							kgitoa_udint(num := kgBatchNoToUDINT(_kgUSINT16toGUID.GUID),str := _sUDINT);
							brsstrcat(ADR(_sSQLstring), ADR(_sUDINT));

						ELSE

							brsstrcat(ADR(_sSQLstring), ADR('@BatchID_GUID = $''));
							_kgGUIDtoSTRING(GUID := _kgUSINT16toGUID.GUID);
							brsstrcat(ADR(_sSQLstring), ADR(_kgGUIDtoSTRING.sOut));
							brsstrcat(ADR(_sSQLstring), ADR('$''));

						END_IF

						brsstrcat(ADR(_sSQLstring), ADR(', @MachineID = N$''));
						brsstrcat(ADR(_sSQLstring), ADR(_sMNo));
						brsstrcat(ADR(_sSQLstring), ADR('$''));

						brsstrcat(ADR(_sSQLstring), ADR(', @CategoryNoAlpha = $''));
						brsstrcat(ADR(_sSQLstring), ADR(IFhlDFII.In.ReqCntBatchEvt.CntBatchEvtList[_bCntWrCntBatchEvt].Batch.sCategory));
						brsstrcat(ADR(_sSQLstring), ADR('$''));

						brsstrcat(ADR(_sSQLstring), ADR(', @ProgNo = '));
						itoa(IFhlDFII.In.ReqCntBatchEvt.CntBatchEvtList[_bCntWrCntBatchEvt].bProgram, ADR(_sValue));
						brsstrcat(ADR(_sSQLstring), ADR(_sValue));

						brsstrcat(ADR(_sSQLstring), ADR(', @Selection = N$''));
						brwcsconv(ADR(_sMark), ADR(IFhlDFII.In.ReqCntBatchEvt.CntBatchEvtList[_bCntWrCntBatchEvt].Batch.utfMark), 1);
						brsstrcat(ADR(_sSQLstring), ADR(_sMark));
						brsstrcat(ADR(_sSQLstring), ADR('$''));

						brsstrcat(ADR(_sSQLstring), ADR(', @Time = $''));
						_mnParam_datetimetoa(dtTimestamp := IFhlDFII.In.ReqCntBatchEvt.CntBatchEvtList[_bCntWrCntBatchEvt].Batch.dtTimeStamp);
						brsstrcat(ADR(_sSQLstring), ADR(_mnParam_datetimetoa.sDateTime));
						brsstrcat(ADR(_sSQLstring), ADR('$'$R$L'));

						IF IFhlDFII.In.ReqCntBatchEvt.CntBatchEvtList[_bCntWrCntBatchEvt].Batch.bCntCustomers > 0 AND IFhlDFII.In.ReqCntBatchEvt.CntBatchEvtList[_bCntWrCntBatchEvt].Batch.bCntCustomers <= 8 THEN

							FOR _ii := 1 TO IFhlDFII.In.ReqCntBatchEvt.CntBatchEvtList[_bCntWrCntBatchEvt].Batch.bCntCustomers DO

								_idxCustomer := _ii - 1;

								brsstrcat(ADR(_sSQLstring), ADR('EXEC [dbo].[spInsEventStatItem_PartBatch] '));

								_kgUSINT16toGUID(usintarray := IFhlDFII.In.ReqCntBatchEvt.CntBatchEvtList[_bCntWrCntBatchEvt].Batch.bBatchNo);

								IF IFhlDFII.In.ReqCntBatchEvt.CntBatchEvtList[_bCntWrCntBatchEvt].Batch.bTypeBatchNo = 0 THEN

									brsstrcat(ADR(_sSQLstring), ADR('@BatchID_INT = '));
									kgitoa_udint(num := kgBatchNoToUDINT(_kgUSINT16toGUID.GUID),str := _sUDINT);
									brsstrcat(ADR(_sSQLstring), ADR(_sUDINT));

								ELSE

									brsstrcat(ADR(_sSQLstring), ADR('@BatchID_GUID = $''));
									_kgGUIDtoSTRING(GUID := _kgUSINT16toGUID.GUID);
									brsstrcat(ADR(_sSQLstring), ADR(_kgGUIDtoSTRING.sOut));
									brsstrcat(ADR(_sSQLstring), ADR('$''));

								END_IF

								brsstrcat(ADR(_sSQLstring), ADR(', @Machine = N$''));
								brsstrcat(ADR(_sSQLstring), ADR(_sMNo));
								brsstrcat(ADR(_sSQLstring), ADR('$''));

								brsstrcat(ADR(_sSQLstring), ADR(', @PartBatchID = '));
								brsitoa(_ii, ADR(_sValue));
								brsstrcat(ADR(_sSQLstring), ADR(_sValue));

								brsstrcat(ADR(_sSQLstring), ADR(', @ActualAmount = '));
								_sValue := REAL_TO_STRING(UINT_TO_REAL(IFhlDFII.In.ReqCntBatchEvt.CntBatchEvtList[_bCntWrCntBatchEvt].Batch.PartBatch[_idxCustomer].wCustomWeight)/10.0);
								brsstrcat(ADR(_sSQLstring), ADR(_sValue));

								brsstrcat(ADR(_sSQLstring), ADR(', @Customer = $''));
								brsstrcat(ADR(_sSQLstring), ADR(IFhlDFII.In.ReqCntBatchEvt.CntBatchEvtList[_bCntWrCntBatchEvt].Batch.PartBatch[_idxCustomer].sCustomNo));
								brsstrcat(ADR(_sSQLstring), ADR('$''));

								IF IFhlDFII.In.ReqCntBatchEvt.CntBatchEvtList[_bCntWrCntBatchEvt].bEvent = MNCNT_BATCHEVENT_LOAD THEN

									brsstrcat(ADR(_sSQLstring), ADR(', @FromOutside = 1, @ToOutside = 0 '));

								END_IF

								IF IFhlDFII.In.ReqCntBatchEvt.CntBatchEvtList[_bCntWrCntBatchEvt].bEvent = MNCNT_BATCHEVENT_UNLOAD THEN

									brsstrcat(ADR(_sSQLstring), ADR(', @FromOutside = 0, @ToOutside = 1  '));

								END_IF

								brsstrcat(ADR(_sSQLstring), ADR(', @FromName = N$''));
								brsstrcat(ADR(_sSQLstring), ADR(IFhlDFII.In.ReqCntBatchEvt.CntBatchEvtList[_bCntWrCntBatchEvt].FromLocation.sNameId));
								brsstrcat(ADR(_sSQLstring), ADR('$''));

								brsstrcat(ADR(_sSQLstring), ADR(', @ToName = N$''));
								brsstrcat(ADR(_sSQLstring), ADR(IFhlDFII.In.ReqCntBatchEvt.CntBatchEvtList[_bCntWrCntBatchEvt].ToLocation.sNameId));
								brsstrcat(ADR(_sSQLstring), ADR('$''));

								brsstrcat(ADR(_sSQLstring), ADR(', @Time = $''));
								_mnParam_datetimetoa(dtTimestamp := IFhlDFII.In.ReqCntBatchEvt.CntBatchEvtList[_bCntWrCntBatchEvt].Batch.dtTimeStamp);
								brsstrcat(ADR(_sSQLstring), ADR(_mnParam_datetimetoa.sDateTime));
								brsstrcat(ADR(_sSQLstring), ADR('$'$R$L'));

							END_FOR

							_DFII_DBExecute.enable := TRUE;
							_DFII_DBExecute.pSqlStatement := ADR(_sSQLstring);
							_DFII_DBExecute.connectionIdent := _lConnectionIdent;

						END_IF

						_sSQLBatchEventString := _sSQLstring;

						_eStep := eSQLREQ_STEP_WRCNTBATCHEVT_r;

					MNCNT_BATCHEVENT_CHANGEDATA:

						_sSQLstring := 'EXEC [dbo].[spUpdEventStat] ';

						_kgUSINT16toGUID(usintarray := IFhlDFII.In.ReqCntBatchEvt.CntBatchEvtList[_bCntWrCntBatchEvt].Batch.bBatchNo);

						IF IFhlDFII.In.ReqCntBatchEvt.CntBatchEvtList[_bCntWrCntBatchEvt].Batch.bTypeBatchNo = 0 THEN

							brsstrcat(ADR(_sSQLstring), ADR('@BatchID_INT = '));
							kgitoa_udint(num := kgBatchNoToUDINT(_kgUSINT16toGUID.GUID),str := _sUDINT);
							brsstrcat(ADR(_sSQLstring), ADR(_sUDINT));

						ELSE

							brsstrcat(ADR(_sSQLstring), ADR('@BatchID_GUID = $''));
							_kgGUIDtoSTRING(GUID := _kgUSINT16toGUID.GUID);
							brsstrcat(ADR(_sSQLstring), ADR(_kgGUIDtoSTRING.sOut));
							brsstrcat(ADR(_sSQLstring), ADR('$''));

						END_IF

						brsstrcat(ADR(_sSQLstring), ADR(', @MachineID = N$''));
						brsstrcat(ADR(_sSQLstring), ADR(_sMNo));
						brsstrcat(ADR(_sSQLstring), ADR('$''));

						brsstrcat(ADR(_sSQLstring), ADR(', @CategoryNoAlpha = $''));
						brsstrcat(ADR(_sSQLstring), ADR(IFhlDFII.In.ReqCntBatchEvt.CntBatchEvtList[_bCntWrCntBatchEvt].Batch.sCategory));
						brsstrcat(ADR(_sSQLstring), ADR('$''));

						brsstrcat(ADR(_sSQLstring), ADR(', @ProgNo = '));
						itoa(IFhlDFII.In.ReqCntBatchEvt.CntBatchEvtList[_bCntWrCntBatchEvt].bProgram, ADR(_sValue));
						brsstrcat(ADR(_sSQLstring), ADR(_sValue));

						brsstrcat(ADR(_sSQLstring), ADR(', @Selection = N$''));
						brwcsconv(ADR(_sMark), ADR(IFhlDFII.In.ReqCntBatchEvt.CntBatchEvtList[_bCntWrCntBatchEvt].Batch.utfMark), 1);
						brsstrcat(ADR(_sSQLstring), ADR(_sMark));
						brsstrcat(ADR(_sSQLstring), ADR('$''));

						brsstrcat(ADR(_sSQLstring), ADR(', @Time = $''));
						_mnParam_datetimetoa(dtTimestamp := IFhlDFII.In.ReqCntBatchEvt.CntBatchEvtList[_bCntWrCntBatchEvt].Batch.dtTimeStamp);
						brsstrcat(ADR(_sSQLstring), ADR(_mnParam_datetimetoa.sDateTime));
						brsstrcat(ADR(_sSQLstring), ADR('$'$R$L'));

						IF IFhlDFII.In.ReqCntBatchEvt.CntBatchEvtList[_bCntWrCntBatchEvt].Batch.bCntCustomers > 0 AND IFhlDFII.In.ReqCntBatchEvt.CntBatchEvtList[_bCntWrCntBatchEvt].Batch.bCntCustomers <= 8 THEN

							FOR _ii := 1 TO IFhlDFII.In.ReqCntBatchEvt.CntBatchEvtList[_bCntWrCntBatchEvt].Batch.bCntCustomers DO

								_idxCustomer := _ii - 1;

								brsstrcat(ADR(_sSQLstring), ADR('EXEC [dbo].[spUpdEventStatItem_PartBatch] '));

								_kgUSINT16toGUID(usintarray := IFhlDFII.In.ReqCntBatchEvt.CntBatchEvtList[_bCntWrCntBatchEvt].Batch.bBatchNo);

								IF IFhlDFII.In.ReqCntBatchEvt.CntBatchEvtList[_bCntWrCntBatchEvt].Batch.bTypeBatchNo = 0 THEN

									brsstrcat(ADR(_sSQLstring), ADR('@BatchID_INT = '));
									kgitoa_udint(num := kgBatchNoToUDINT(_kgUSINT16toGUID.GUID),str := _sUDINT);
									brsstrcat(ADR(_sSQLstring), ADR(_sUDINT));

								ELSE

									brsstrcat(ADR(_sSQLstring), ADR('@BatchID_GUID = $''));
									_kgGUIDtoSTRING(GUID := _kgUSINT16toGUID.GUID);
									brsstrcat(ADR(_sSQLstring), ADR(_kgGUIDtoSTRING.sOut));
									brsstrcat(ADR(_sSQLstring), ADR('$''));

								END_IF

								brsstrcat(ADR(_sSQLstring), ADR(', @Machine = N$''));
								brsstrcat(ADR(_sSQLstring), ADR(_sMNo));
								brsstrcat(ADR(_sSQLstring), ADR('$''));

								brsstrcat(ADR(_sSQLstring), ADR(', @PartBatchID = '));
								brsitoa(_ii, ADR(_sValue));
								brsstrcat(ADR(_sSQLstring), ADR(_sValue));

								brsstrcat(ADR(_sSQLstring), ADR(', @ActualAmount = '));
								_sValue := REAL_TO_STRING(UINT_TO_REAL(IFhlDFII.In.ReqCntBatchEvt.CntBatchEvtList[_bCntWrCntBatchEvt].Batch.PartBatch[_idxCustomer].wCustomWeight)/10.0);
								brsstrcat(ADR(_sSQLstring), ADR(_sValue));

								brsstrcat(ADR(_sSQLstring), ADR(', @Customer = $''));
								brsstrcat(ADR(_sSQLstring), ADR(IFhlDFII.In.ReqCntBatchEvt.CntBatchEvtList[_bCntWrCntBatchEvt].Batch.PartBatch[_idxCustomer].sCustomNo));
								brsstrcat(ADR(_sSQLstring), ADR('$''));

								brsstrcat(ADR(_sSQLstring), ADR(', @Time = $''));
								_mnParam_datetimetoa(dtTimestamp := IFhlDFII.In.ReqCntBatchEvt.CntBatchEvtList[_bCntWrCntBatchEvt].Batch.dtTimeStamp);
								brsstrcat(ADR(_sSQLstring), ADR(_mnParam_datetimetoa.sDateTime));
								brsstrcat(ADR(_sSQLstring), ADR('$'$R$L'));

							END_FOR

							_DFII_DBExecute.enable := TRUE;
							_DFII_DBExecute.pSqlStatement := ADR(_sSQLstring);
							_DFII_DBExecute.connectionIdent := _lConnectionIdent;

						END_IF

						_sSQLBatchEventString := _sSQLstring;

						_eStep := eSQLREQ_STEP_WRCNTBATCHEVT_r;

					MNCNT_BATCHEVENT_DELETE:

						_bCntWrCntBatchEvt := _bCntWrCntBatchEvt + 1;

				END_CASE

			END_IF

		eSQLREQ_STEP_WRCNTBATCHEVT_r:

			_DFII_DBExecute();

			IF _DFII_DBExecute.status = ERR_OK  OR _DFII_DBExecute.dbError = DB_SQL_NO_DATA THEN

				_sLogEntryI := WSTRING_TO_STRING(IFmnParam.Out.utfMachineNumber);
				_sLogEntryI := CONCAT(_sLogEntryI, '-hlDFII$tSUCC$tWRITE BATCH EVENT');
				_InsertRB(wPtrWrite := _wPtrRBwrite, wPtrRead := _wPtrRBread, wPtrStart := _wPtrRBstart);

				_bCntWrCntBatchEvt := _bCntWrCntBatchEvt + 1;
				_eStep := eSQLREQ_STEP_WRCNTBATCHEVT;

			ELSIF _DFII_DBExecute.status <> ERR_FUB_BUSY THEN

				_sAction := 'Write Batch failed:';
				_eStep := eSQLREQ_STEP_GET_ERROR;

			END_IF

		eSQLREQ_STEP_WRCNTCNTEVT:

			IF _bCntWrCntCntEvt > IFhlDFII.In.ReqCntCntEvt.bCntLines THEN

				_eStep := eSQLREQ_STEP_WAITFORCOMMAND;

			ELSE

				CASE IFhlDFII.In.ReqCntCntEvt.CntCounterEvtList[_bCntWrCntCntEvt].bType OF

					MNCNT_COUNTERTYPE_WATER:

						_sSQLstring := 'EXEC [dbo].[spInsEventStatItem_Water] ';

						brsstrcat(ADR(_sSQLstring), ADR('@Machine = N$''));
						brsstrcat(ADR(_sSQLstring), ADR(_sMNo));
						brsstrcat(ADR(_sSQLstring), ADR('$''));

						_kgUSINT16toGUID(usintarray := IFhlDFII.In.ReqCntCntEvt.CntCounterEvtList[_bCntWrCntCntEvt].BatchNo);

						IF NOT kgGUIDisZero(_kgUSINT16toGUID.GUID) THEN

							IF IFhlDFII.In.ReqCntCntEvt.CntCounterEvtList[_bCntWrCntCntEvt].bTypeBatchNo = 0 THEN

								brsstrcat(ADR(_sSQLstring), ADR(', @BatchID_INT = '));
								kgitoa_udint(num := kgBatchNoToUDINT(_kgUSINT16toGUID.GUID),str := _sUDINT);
								brsstrcat(ADR(_sSQLstring), ADR(_sUDINT));

							ELSE

								brsstrcat(ADR(_sSQLstring), ADR(', @BatchID_GUID = $''));
								_kgGUIDtoSTRING(GUID := _kgUSINT16toGUID.GUID);
								brsstrcat(ADR(_sSQLstring), ADR(_kgGUIDtoSTRING.sOut));
								brsstrcat(ADR(_sSQLstring), ADR('$''));

							END_IF

						END_IF

						brsstrcat(ADR(_sSQLstring), ADR(', @ActualAmount = '));
						_sValue := REAL_TO_STRING(UDINT_TO_REAL(IFhlDFII.In.ReqCntCntEvt.CntCounterEvtList[_bCntWrCntCntEvt].lAmount));
						brsstrcat(ADR(_sSQLstring), ADR(_sValue));

						brsstrcat(ADR(_sSQLstring), ADR(', @TargetAmount = '));
						_sValue := REAL_TO_STRING(UDINT_TO_REAL(IFhlDFII.In.ReqCntCntEvt.CntCounterEvtList[_bCntWrCntCntEvt].lNomAmount));
						brsstrcat(ADR(_sSQLstring), ADR(_sValue));

						//							IF IFhlDFII.In.ReqCntCntEvt.CntCounterEvtList[_bCntWrCntCntEvt].Source.bCompartment > 0 THEN
						//
						//								brsstrcat(ADR(_sSQLstring), ADR(', @FromChamber = '));
						//								_sValue := USINT_TO_STRING(IFhlDFII.In.ReqCntCntEvt.CntCounterEvtList[_bCntWrCntCntEvt].Source.bCompartment);
						//								brsstrcat(ADR(_sSQLstring), ADR(_sValue));
						//
						//							ELSE

						brsstrcat(ADR(_sSQLstring), ADR(', @FromName = N$''));
						brsstrcat(ADR(_sSQLstring), ADR(IFhlDFII.In.ReqCntCntEvt.CntCounterEvtList[_bCntWrCntCntEvt].Source.sNameId));
						brsstrcat(ADR(_sSQLstring), ADR('$''));

						//							END_IF

						IF IFhlDFII.In.ReqCntCntEvt.CntCounterEvtList[_bCntWrCntCntEvt].Source.bLocationExt > 0 THEN

							brsstrcat(ADR(_sSQLstring), ADR(', @FromOutside = 1'));

						ELSE

							brsstrcat(ADR(_sSQLstring), ADR(', @FromOutside = 0'));

						END_IF

						//							IF IFhlDFII.In.ReqCntCntEvt.CntCounterEvtList[_bCntWrCntCntEvt].Destination.bCompartment > 0 THEN
						//
						//								brsstrcat(ADR(_sSQLstring), ADR(', @ToChamber = '));
						//								_sValue := USINT_TO_STRING(IFhlDFII.In.ReqCntCntEvt.CntCounterEvtList[_bCntWrCntCntEvt].Destination.bCompartment);
						//								brsstrcat(ADR(_sSQLstring), ADR(_sValue));
						//
						//							ELSE

						brsstrcat(ADR(_sSQLstring), ADR(', @ToName = N$''));
						brsstrcat(ADR(_sSQLstring), ADR(IFhlDFII.In.ReqCntCntEvt.CntCounterEvtList[_bCntWrCntCntEvt].Destination.sNameId));
						brsstrcat(ADR(_sSQLstring), ADR('$''));

						//							END_IF

						IF IFhlDFII.In.ReqCntCntEvt.CntCounterEvtList[_bCntWrCntCntEvt].Destination.bLocationExt > 0 THEN

							brsstrcat(ADR(_sSQLstring), ADR(', @ToOutside = 1'));

						ELSE

							brsstrcat(ADR(_sSQLstring), ADR(', @ToOutside = 0'));

						END_IF

						brsstrcat(ADR(_sSQLstring), ADR(', @Time = $''));
						_mnParam_datetimetoa(dtTimestamp := IFhlDFII.In.ReqCntCntEvt.CntCounterEvtList[_bCntWrCntCntEvt].dtTimeStamp);
						brsstrcat(ADR(_sSQLstring), ADR(_mnParam_datetimetoa.sDateTime));
						brsstrcat(ADR(_sSQLstring), ADR('$''));

						_DFII_DBExecute.enable := TRUE;
						_DFII_DBExecute.pSqlStatement := ADR(_sSQLstring);
						_DFII_DBExecute.connectionIdent := _lConnectionIdent;

						_eStep := eSQLREQ_STEP_WRCNTCNTEVT_r;

					MNCNT_COUNTERTYPE_TEMPERATURE:

						_sSQLstring := 'EXEC [dbo].[spInsEventStatItem_Temperature] ';

						brsstrcat(ADR(_sSQLstring), ADR('@Machine = N$''));
						brsstrcat(ADR(_sSQLstring), ADR(_sMNo));
						brsstrcat(ADR(_sSQLstring), ADR('$''));

						_kgUSINT16toGUID(usintarray := IFhlDFII.In.ReqCntCntEvt.CntCounterEvtList[_bCntWrCntCntEvt].BatchNo);

						IF NOT kgGUIDisZero(_kgUSINT16toGUID.GUID) THEN

							IF IFhlDFII.In.ReqCntCntEvt.CntCounterEvtList[_bCntWrCntCntEvt].bTypeBatchNo = 0 THEN

								brsstrcat(ADR(_sSQLstring), ADR(', @BatchID_INT = '));
								kgitoa_udint(num := kgBatchNoToUDINT(_kgUSINT16toGUID.GUID),str := _sUDINT);
								brsstrcat(ADR(_sSQLstring), ADR(_sUDINT));

							ELSE

								brsstrcat(ADR(_sSQLstring), ADR(', @BatchID_GUID = $''));
								_kgGUIDtoSTRING(GUID := _kgUSINT16toGUID.GUID);
								brsstrcat(ADR(_sSQLstring), ADR(_kgGUIDtoSTRING.sOut));
								brsstrcat(ADR(_sSQLstring), ADR('$''));

							END_IF

						END_IF

						brsstrcat(ADR(_sSQLstring), ADR(', @ActualAmount = '));
						_sValue := REAL_TO_STRING(UDINT_TO_REAL(IFhlDFII.In.ReqCntCntEvt.CntCounterEvtList[_bCntWrCntCntEvt].lAmount));
						brsstrcat(ADR(_sSQLstring), ADR(_sValue));

						brsstrcat(ADR(_sSQLstring), ADR(', @TargetAmount = '));
						_sValue := REAL_TO_STRING(UDINT_TO_REAL(IFhlDFII.In.ReqCntCntEvt.CntCounterEvtList[_bCntWrCntCntEvt].lNomAmount));
						brsstrcat(ADR(_sSQLstring), ADR(_sValue));

						//							IF IFhlDFII.In.ReqCntCntEvt.CntCounterEvtList[_bCntWrCntCntEvt].Destination.bCompartment > 0 THEN
						//
						//								brsstrcat(ADR(_sSQLstring), ADR(', @LocationChamber = '));
						//								_sValue := USINT_TO_STRING(IFhlDFII.In.ReqCntCntEvt.CntCounterEvtList[_bCntWrCntCntEvt].Destination.bCompartment);
						//								brsstrcat(ADR(_sSQLstring), ADR(_sValue));
						//
						//							ELSE

						brsstrcat(ADR(_sSQLstring), ADR(', @LocationName = N$''));
						brsstrcat(ADR(_sSQLstring), ADR(IFhlDFII.In.ReqCntCntEvt.CntCounterEvtList[_bCntWrCntCntEvt].Destination.sNameId));
						brsstrcat(ADR(_sSQLstring), ADR('$''));

						//							END_IF

						IF IFhlDFII.In.ReqCntCntEvt.CntCounterEvtList[_bCntWrCntCntEvt].Destination.bLocationExt > 0 THEN

							brsstrcat(ADR(_sSQLstring), ADR(', @LocationOutside = 1'));

						ELSE

							brsstrcat(ADR(_sSQLstring), ADR(', @LocationOutside = 0'));

						END_IF

						brsstrcat(ADR(_sSQLstring), ADR(', @Time = $''));
						_mnParam_datetimetoa(dtTimestamp := IFhlDFII.In.ReqCntCntEvt.CntCounterEvtList[_bCntWrCntCntEvt].dtTimeStamp);
						brsstrcat(ADR(_sSQLstring), ADR(_mnParam_datetimetoa.sDateTime));
						brsstrcat(ADR(_sSQLstring), ADR('$''));

						_DFII_DBExecute.enable := TRUE;
						_DFII_DBExecute.pSqlStatement := ADR(_sSQLstring);
						_DFII_DBExecute.connectionIdent := _lConnectionIdent;

						_eStep := eSQLREQ_STEP_WRCNTCNTEVT_r;

					MNCNT_COUNTERTYPE_STEAM, MNCNT_COUNTERTYPE_ELECTRICENERGY, MNCNT_COUNTERTYPE_GAS:

						IF IFhlDFII.In.ReqCntCntEvt.CntCounterEvtList[_bCntWrCntCntEvt].bType = MNCNT_COUNTERTYPE_STEAM THEN
							_sSQLstring := 'EXEC [dbo].[spInsEventStatItem_Steam] ';
						ELSIF IFhlDFII.In.ReqCntCntEvt.CntCounterEvtList[_bCntWrCntCntEvt].bType = MNCNT_COUNTERTYPE_GAS THEN
							_sSQLstring := 'EXEC [dbo].[spInsEventStatItem_Gas] ';
						ELSE
							_sSQLstring := 'EXEC [dbo].[spInsEventStatItem_Energy] ';
						END_IF

						brsstrcat(ADR(_sSQLstring), ADR('@Machine = N$''));
						brsstrcat(ADR(_sSQLstring), ADR(_sMNo));
						brsstrcat(ADR(_sSQLstring), ADR('$''));

						_kgUSINT16toGUID(usintarray := IFhlDFII.In.ReqCntCntEvt.CntCounterEvtList[_bCntWrCntCntEvt].BatchNo);

						IF NOT kgGUIDisZero(_kgUSINT16toGUID.GUID) THEN

							IF IFhlDFII.In.ReqCntCntEvt.CntCounterEvtList[_bCntWrCntCntEvt].bTypeBatchNo = 0 THEN

								brsstrcat(ADR(_sSQLstring), ADR(', @BatchID_INT = '));
								kgitoa_udint(num := kgBatchNoToUDINT(_kgUSINT16toGUID.GUID),str := _sUDINT);
								brsstrcat(ADR(_sSQLstring), ADR(_sUDINT));

							ELSE

								brsstrcat(ADR(_sSQLstring), ADR(', @BatchID_GUID = $''));
								_kgGUIDtoSTRING(GUID := _kgUSINT16toGUID.GUID);
								brsstrcat(ADR(_sSQLstring), ADR(_kgGUIDtoSTRING.sOut));
								brsstrcat(ADR(_sSQLstring), ADR('$''));

							END_IF

						END_IF

						brsstrcat(ADR(_sSQLstring), ADR(', @ActualAmount = '));
						_sValue := REAL_TO_STRING(UDINT_TO_REAL(IFhlDFII.In.ReqCntCntEvt.CntCounterEvtList[_bCntWrCntCntEvt].lAmount));
						brsstrcat(ADR(_sSQLstring), ADR(_sValue));

						//							IF IFhlDFII.In.ReqCntCntEvt.CntCounterEvtList[_bCntWrCntCntEvt].Source.bCompartment > 0 THEN
						//
						//								brsstrcat(ADR(_sSQLstring), ADR(', @FromChamber = '));
						//								_sValue := USINT_TO_STRING(IFhlDFII.In.ReqCntCntEvt.CntCounterEvtList[_bCntWrCntCntEvt].Source.bCompartment);
						//								brsstrcat(ADR(_sSQLstring), ADR(_sValue));
						//
						//							ELSE

						brsstrcat(ADR(_sSQLstring), ADR(', @FromName = N$''));
						brsstrcat(ADR(_sSQLstring), ADR(IFhlDFII.In.ReqCntCntEvt.CntCounterEvtList[_bCntWrCntCntEvt].Source.sNameId));
						brsstrcat(ADR(_sSQLstring), ADR('$''));

						//							END_IF

						IF IFhlDFII.In.ReqCntCntEvt.CntCounterEvtList[_bCntWrCntCntEvt].Source.bLocationExt > 0 THEN

							brsstrcat(ADR(_sSQLstring), ADR(', @FromOutside = 1'));

						ELSE

							brsstrcat(ADR(_sSQLstring), ADR(', @FromOutside = 0'));

						END_IF

						//							IF IFhlDFII.In.ReqCntCntEvt.CntCounterEvtList[_bCntWrCntCntEvt].Destination.bCompartment > 0 THEN
						//
						//								brsstrcat(ADR(_sSQLstring), ADR(', @ToChamber = '));
						//								_sValue := USINT_TO_STRING(IFhlDFII.In.ReqCntCntEvt.CntCounterEvtList[_bCntWrCntCntEvt].Destination.bCompartment);
						//								brsstrcat(ADR(_sSQLstring), ADR(_sValue));
						//
						//							ELSE

						brsstrcat(ADR(_sSQLstring), ADR(', @ToName = N$''));
						brsstrcat(ADR(_sSQLstring), ADR(IFhlDFII.In.ReqCntCntEvt.CntCounterEvtList[_bCntWrCntCntEvt].Destination.sNameId));
						brsstrcat(ADR(_sSQLstring), ADR('$''));

						//							END_IF

						IF IFhlDFII.In.ReqCntCntEvt.CntCounterEvtList[_bCntWrCntCntEvt].Destination.bLocationExt > 0 THEN

							brsstrcat(ADR(_sSQLstring), ADR(', @ToOutside = 1'));

						ELSE

							brsstrcat(ADR(_sSQLstring), ADR(', @ToOutside = 0'));

						END_IF

						brsstrcat(ADR(_sSQLstring), ADR(', @Time = $''));
						_mnParam_datetimetoa(dtTimestamp := IFhlDFII.In.ReqCntCntEvt.CntCounterEvtList[_bCntWrCntCntEvt].dtTimeStamp);
						brsstrcat(ADR(_sSQLstring), ADR(_mnParam_datetimetoa.sDateTime));
						brsstrcat(ADR(_sSQLstring), ADR('$''));

						_DFII_DBExecute.enable := TRUE;
						_DFII_DBExecute.pSqlStatement := ADR(_sSQLstring);
						_DFII_DBExecute.connectionIdent := _lConnectionIdent;

						_eStep := eSQLREQ_STEP_WRCNTCNTEVT_r;

					ELSE

						_bCntWrCntCntEvt := _bCntWrCntCntEvt + 1;

				END_CASE

			END_IF

		eSQLREQ_STEP_WRCNTCNTEVT_r:

			_DFII_DBExecute();

			IF _DFII_DBExecute.status = ERR_OK  OR _DFII_DBExecute.dbError = DB_SQL_NO_DATA THEN

				_sLogEntryI := WSTRING_TO_STRING(IFmnParam.Out.utfMachineNumber);
				_sLogEntryI := CONCAT(_sLogEntryI, '-hlDFII$tSUCC$tWRITE COUNT EVENT');
				_InsertRB(wPtrWrite := _wPtrRBwrite, wPtrRead := _wPtrRBread, wPtrStart := _wPtrRBstart);

				_bCntWrCntCntEvt := _bCntWrCntCntEvt + 1;
				_eStep := eSQLREQ_STEP_WRCNTCNTEVT;

			ELSIF _DFII_DBExecute.status <> ERR_FUB_BUSY THEN

				_sAction := 'Write Counter failed:';
				_eStep := eSQLREQ_STEP_GET_ERROR;

			END_IF

		// Zeitzähler senden

		eSQLREQ_STEP_WRCNTTIMEVT:

			IF _bCntWrCntTimeEvt > IFhlDFII.In.ReqCntTimEvt.bCntLines THEN

				_eStep := eSQLREQ_STEP_WAITFORCOMMAND;

			ELSE

				_sSQLstring := 'EXEC [dbo].[spInsEventStatItem_StateTime] ';

				brsstrcat(ADR(_sSQLstring), ADR('@Machine = N$''));
				brsstrcat(ADR(_sSQLstring), ADR(_sMNo));
				brsstrcat(ADR(_sSQLstring), ADR('$''));

				brsstrcat(ADR(_sSQLstring), ADR(', @ActualAmount = '));
				_sValue := REAL_TO_STRING(UDINT_TO_REAL(IFhlDFII.In.ReqCntTimEvt.CntTimerEvtList[_bCntWrCntTimeEvt].lAmount));
				brsstrcat(ADR(_sSQLstring), ADR(_sValue));

				IF IFhlDFII.In.ReqCntTimEvt.CntTimerEvtList[_bCntWrCntTimeEvt].bState = MNCNT_TIMERSTATE_PAUSED THEN

					brsstrcat(ADR(_sSQLstring), ADR(', @State = $'PAUSED$''));

					CASE IFhlDFII.In.ReqCntTimEvt.CntTimerEvtList[_bCntWrCntTimeEvt].bSubState OF

						MNCNT_TIMERSUBSTATE_OFF:

							brsstrcat(ADR(_sSQLstring), ADR(', @SubState = $'OFF$''));

						MNCNT_TIMERSUBSTATE_STOP:

							brsstrcat(ADR(_sSQLstring), ADR(', @SubState = $'STOP$''));

						MNCNT_TIMERSUBSTATE_INTFAULT:

							brsstrcat(ADR(_sSQLstring), ADR(', @SubState = $'INTFAULT$''));

						MNCNT_TIMERSUBSTATE_EXTFAULT:

							brsstrcat(ADR(_sSQLstring), ADR(', @SubState = $'EXTFAULT$''));

						MNCNT_TIMERSUBSTATE_SAFESTOP:

							brsstrcat(ADR(_sSQLstring), ADR(', @SubState = $'SAFESTOP$''));

						MNCNT_TIMERSUBSTATE_EMERGENCYSTP:

							brsstrcat(ADR(_sSQLstring), ADR(', @SubState = $'EMERGSTOP$''));

						ELSE

							brsstrcat(ADR(_sSQLstring), ADR(', @SubState = $'$''));

					END_CASE

				ELSIF IFhlDFII.In.ReqCntTimEvt.CntTimerEvtList[_bCntWrCntTimeEvt].bState = MNCNT_TIMERSTATE_WAIT THEN

					brsstrcat(ADR(_sSQLstring), ADR(', @State = $'WAIT$''));

					CASE IFhlDFII.In.ReqCntTimEvt.CntTimerEvtList[_bCntWrCntTimeEvt].bSubState OF

						MNCNT_TIMERSUBSTATE_LOADING:

							brsstrcat(ADR(_sSQLstring), ADR(', @SubState = $'LOADING$''));

						MNCNT_TIMERSUBSTATE_UNLOADING:

							brsstrcat(ADR(_sSQLstring), ADR(', @SubState = $'UNLOADING$''));

						MNCNT_TIMERSUBSTATE_DOSING:

							brsstrcat(ADR(_sSQLstring), ADR(', @SubState = $'DOSING$''));

						MNCNT_TIMERSUBSTATE_WATERLEVEL:

							brsstrcat(ADR(_sSQLstring), ADR(', @SubState = $'WATERLEVEL$''));

						MNCNT_TIMERSUBSTATE_TEMPERATURE:

							brsstrcat(ADR(_sSQLstring), ADR(', @SubState = $'TEMP$''));

						MNCNT_TIMERSUBSTATE_DISINFECTION:

							brsstrcat(ADR(_sSQLstring), ADR(', @SubState = $'DISINFECT$''));

						MNCNT_TIMERSUBSTATE_AIRPRESSURE:

							brsstrcat(ADR(_sSQLstring), ADR(', @SubState = $'AIRPRESS$''));

						ELSE

							brsstrcat(ADR(_sSQLstring), ADR(', @SubState = $'$''));

					END_CASE

				ELSIF IFhlDFII.In.ReqCntTimEvt.CntTimerEvtList[_bCntWrCntTimeEvt].bState = MNCNT_TIMERSTATE_ACTIVE THEN

					brsstrcat(ADR(_sSQLstring), ADR(', @State = $'ACTIVE$''));

					CASE IFhlDFII.In.ReqCntTimEvt.CntTimerEvtList[_bCntWrCntTimeEvt].bSubState OF

						MNCNT_TIMERSUBSTATE_WASHING:

							brsstrcat(ADR(_sSQLstring), ADR(', @SubState = $'PROCESSING$''));

						MNCNT_TIMERSUBSTATE_PREPERATION:

							brsstrcat(ADR(_sSQLstring), ADR(', @SubState = $'PREP$''));

						MNCNT_TIMERSUBSTATE_TRANSFER:

							brsstrcat(ADR(_sSQLstring), ADR(', @SubState = $'TRANSFER$''));

						MNCNT_TIMERSUBSTATE_PREPFORSTOP:

							brsstrcat(ADR(_sSQLstring), ADR(', @SubState = $'PREPFORSTOP$''));

						ELSE

							brsstrcat(ADR(_sSQLstring), ADR(', @SubState = $'$''));

					END_CASE

				ELSE

					brsstrcat(ADR(_sSQLstring), ADR(', @State = $'$', @SubState = $'$''));

				END_IF

				brsstrcat(ADR(_sSQLstring), ADR(', @Time = $''));
				_mnParam_datetimetoa(dtTimestamp := IFhlDFII.In.ReqCntTimEvt.CntTimerEvtList[_bCntWrCntTimeEvt].dtTimeStamp);
				brsstrcat(ADR(_sSQLstring), ADR(_mnParam_datetimetoa.sDateTime));
				brsstrcat(ADR(_sSQLstring), ADR('$''));

				_DFII_DBExecute.enable := TRUE;
				_DFII_DBExecute.pSqlStatement := ADR(_sSQLstring);
				_DFII_DBExecute.connectionIdent := _lConnectionIdent;

				_eStep := eSQLREQ_STEP_WRCNTTIMEVT_r;

			END_IF

		eSQLREQ_STEP_WRCNTTIMEVT_r:

			_DFII_DBExecute();

			IF _DFII_DBExecute.status = ERR_OK  OR _DFII_DBExecute.dbError = DB_SQL_NO_DATA THEN

				_sLogEntryI := WSTRING_TO_STRING(IFmnParam.Out.utfMachineNumber);
				_sLogEntryI := CONCAT(_sLogEntryI, '-hlDFII$tSUCC$tWRITE TIME EVENT');
				_InsertRB(wPtrWrite := _wPtrRBwrite, wPtrRead := _wPtrRBread, wPtrStart := _wPtrRBstart);

				_bCntWrCntTimeEvt := _bCntWrCntTimeEvt + 1;
				_eStep := eSQLREQ_STEP_WRCNTTIMEVT;

			ELSIF _DFII_DBExecute.status <> ERR_FUB_BUSY THEN

				_sAction := 'Write Time failed:';
				_eStep := eSQLREQ_STEP_GET_ERROR;

			END_IF

		// Dosierevents schreiben

		eSQLREQ_STEP_WRCNTDOSEVT:

			IF _bCntWrCntDoseEvt > IFhlDFII.In.ReqCntDosEvt.bCntLines THEN

				_eStep := eSQLREQ_STEP_WAITFORCOMMAND;

			ELSE

				_sSQLstring := 'EXEC [dbo].[spInsEventStatItem_Chemical] ';

				brsstrcat(ADR(_sSQLstring), ADR('@Machine = N$''));
				brsstrcat(ADR(_sSQLstring), ADR(_sMNo));
				brsstrcat(ADR(_sSQLstring), ADR('$''));

				_kgUSINT16toGUID(usintarray := IFhlDFII.In.ReqCntDosEvt.CntDosingEvtList[_bCntWrCntDoseEvt].DosingEvent.BatchNo);

				IF NOT kgGUIDisZero(_kgUSINT16toGUID.GUID) THEN

					IF IFhlDFII.In.ReqCntDosEvt.CntDosingEvtList[_bCntWrCntDoseEvt].DosingEvent.bTypeBatchNo = 0 THEN

						brsstrcat(ADR(_sSQLstring), ADR(', @BatchID_INT = '));
						kgitoa_udint(num := kgBatchNoToUDINT(_kgUSINT16toGUID.GUID),str := _sUDINT);
						brsstrcat(ADR(_sSQLstring), ADR(_sUDINT));

					ELSE

						brsstrcat(ADR(_sSQLstring), ADR(', @BatchID_GUID = $''));
						_kgGUIDtoSTRING(GUID := _kgUSINT16toGUID.GUID);
						brsstrcat(ADR(_sSQLstring), ADR(_kgGUIDtoSTRING.sOut));
						brsstrcat(ADR(_sSQLstring), ADR('$''));

					END_IF

				END_IF

				brsstrcat(ADR(_sSQLstring), ADR(', @ActualAmount = '));
				_sValue := REAL_TO_STRING(IFhlDFII.In.ReqCntDosEvt.CntDosingEvtList[_bCntWrCntDoseEvt].DosingEvent.rAmount);
				brsstrcat(ADR(_sSQLstring), ADR(_sValue));

				brsstrcat(ADR(_sSQLstring), ADR(', @TargetAmount = '));
				_sValue := REAL_TO_STRING(IFhlDFII.In.ReqCntDosEvt.CntDosingEvtList[_bCntWrCntDoseEvt].DosingEvent.rNomAmount);
				brsstrcat(ADR(_sSQLstring), ADR(_sValue));

				brsstrcat(ADR(_sSQLstring), ADR(', @Unit = $''));
				brsstrcat(ADR(_sSQLstring), ADR(IFhlDFII.In.ReqCntDosEvt.CntDosingEvtList[_bCntWrCntDoseEvt].DosingEvent.sUnit));
				brsstrcat(ADR(_sSQLstring), ADR('$''));

				_sDoseName := WSTRING_TO_STRING(IFhlDFII.In.ReqCntDosEvt.CntDosingEvtList[_bCntWrCntDoseEvt].DosingEvent.utfName);

				brsstrcat(ADR(_sSQLstring), ADR(', @Name = N$''));
				brsstrcat(ADR(_sSQLstring), ADR(_sDoseName));
				brsstrcat(ADR(_sSQLstring), ADR('$''));

				brsstrcat(ADR(_sSQLstring), ADR(', @FromName = N$''));
				brsstrcat(ADR(_sSQLstring), ADR(IFhlDFII.In.ReqCntDosEvt.CntDosingEvtList[_bCntWrCntDoseEvt].DosingEvent.Source.sNameId));
				brsstrcat(ADR(_sSQLstring), ADR('$''));

				IF IFhlDFII.In.ReqCntDosEvt.CntDosingEvtList[_bCntWrCntDoseEvt].DosingEvent.Source.bLocationExt > 0 THEN

					brsstrcat(ADR(_sSQLstring), ADR(', @FromOutside = 1'));

				ELSE

					brsstrcat(ADR(_sSQLstring), ADR(', @FromOutside = 0'));

				END_IF

				brsstrcat(ADR(_sSQLstring), ADR(', @ToName = N$''));
				brsstrcat(ADR(_sSQLstring), ADR(IFhlDFII.In.ReqCntDosEvt.CntDosingEvtList[_bCntWrCntDoseEvt].DosingEvent.Destination.sNameId));
				brsstrcat(ADR(_sSQLstring), ADR('$''));

				IF IFhlDFII.In.ReqCntDosEvt.CntDosingEvtList[_bCntWrCntDoseEvt].DosingEvent.Destination.bLocationExt > 0 THEN

					brsstrcat(ADR(_sSQLstring), ADR(', @ToOutside = 1'));

				ELSE

					brsstrcat(ADR(_sSQLstring), ADR(', @ToOutside = 0'));

				END_IF

				brsstrcat(ADR(_sSQLstring), ADR(', @Time = $''));
				_mnParam_datetimetoa(dtTimestamp := IFhlDFII.In.ReqCntDosEvt.CntDosingEvtList[_bCntWrCntDoseEvt].DosingEvent.dtTimeStamp);
				brsstrcat(ADR(_sSQLstring), ADR(_mnParam_datetimetoa.sDateTime));
				brsstrcat(ADR(_sSQLstring), ADR('$''));

				_DFII_DBExecute.enable := TRUE;
				_DFII_DBExecute.pSqlStatement := ADR(_sSQLstring);
				_DFII_DBExecute.connectionIdent := _lConnectionIdent;

				_eStep := eSQLREQ_STEP_WRCNTDOSEVT_r;

			END_IF

		eSQLREQ_STEP_WRCNTDOSEVT_r:

			_DFII_DBExecute();

			IF _DFII_DBExecute.status = ERR_OK  OR _DFII_DBExecute.dbError = DB_SQL_NO_DATA THEN

				_sLogEntryI := WSTRING_TO_STRING(IFmnParam.Out.utfMachineNumber);
				_sLogEntryI := CONCAT(_sLogEntryI, '-hlDFII$tSUCC$tWRITE DOSING EVENT');
				_InsertRB(wPtrWrite := _wPtrRBwrite, wPtrRead := _wPtrRBread, wPtrStart := _wPtrRBstart);

				_bCntWrCntDoseEvt := _bCntWrCntDoseEvt + 1;
				_eStep := eSQLREQ_STEP_WRCNTDOSEVT;

			ELSIF _DFII_DBExecute.status <> ERR_FUB_BUSY THEN

				_sAction := 'Write Dosing failed:';
				_eStep := eSQLREQ_STEP_GET_ERROR;

			END_IF

		// Maschine registrieren
		eSQLREQ_STEP_REGMACH:

			brsstrcpy(ADR(_sSQLstring), ADR('EXEC [dbo].[spRegMachine01]  @MachineID = N$''));
			brsstrcat(ADR(_sSQLstring), ADR(_sMNo));
			brsstrcat(ADR(_sSQLstring), ADR('$''));

			brsstrcat(ADR(_sSQLstring),ADR(', @ShortName = $''));
			brwcsconv(ADR(_sShortName),ADR(mnParamStatAd.HeaderVersion.utfMachineType),1);
			brsstrcat(ADR(_sSQLstring),ADR(_sShortName));
			brsstrcat(ADR(_sSQLstring),ADR('$''));

			brsstrcat(ADR(_sSQLstring),ADR(', @Name = $''));
			brwcsconv(ADR(_sName),ADR(mnParamStatAd.utfMachineName),1);
			brsstrcat(ADR(_sSQLstring),ADR(_sName));
			brsstrcat(ADR(_sSQLstring),ADR('$''));

			_DFII_DBExecute.enable := TRUE;
			_DFII_DBExecute.pSqlStatement := ADR(_sSQLstring);
			_DFII_DBExecute.connectionIdent := _lConnectionIdent;

			_eStep := eSQLREQ_STEP_REGMACH_r;

		eSQLREQ_STEP_REGMACH_r:

			_DFII_DBExecute();

			IF _DFII_DBExecute.status = ERR_OK  OR _DFII_DBExecute.dbError = DB_SQL_NO_DATA THEN

				_sLogEntryI := WSTRING_TO_STRING(IFmnParam.Out.utfMachineNumber);
				_sLogEntryI := CONCAT(_sLogEntryI, '-hlDFII$tSUCC$tREGMACHINE');
				_InsertRB(wPtrWrite := _wPtrRBwrite, wPtrRead := _wPtrRBread, wPtrStart := _wPtrRBstart);

				_eStep := eSQLREQ_STEP_WAITFORCOMMAND;

			ELSIF _DFII_DBExecute.status <> ERR_FUB_BUSY THEN

				_sAction := 'Reg. Machine failed:';
				_eStep := eSQLREQ_STEP_GET_ERROR;

			END_IF

		// Uhrzeit von DB lesen
		eSQLREQ_STEP_GETTIME:

			_sSQLstring := 'SELECT DATEDIFF(s,$'1970-01-01T00:00:00$',GETDATE())';

			_DFII_DBExecute.enable := TRUE;
			_DFII_DBExecute.pSqlStatement := ADR(_sSQLstring);
			_DFII_DBExecute.connectionIdent := _lConnectionIdent;

			_eStep := eSQLREQ_STEP_GETTIME_r;

		eSQLREQ_STEP_GETTIME_r:

			_DFII_DBExecute();

			IF _DFII_DBExecute.status = ERR_OK THEN

				_eStep := eSQLREQ_STEP_GETTIME_FETCH;

			ELSIF _DFII_DBExecute.status <> ERR_FUB_BUSY THEN

				_sAction := 'Get Time failed:';
				_eStep := eSQLREQ_STEP_GET_ERROR;

			END_IF

		(* Zeile holen *)
		eSQLREQ_STEP_GETTIME_FETCH:

			_DFII_DBFetch.enable := TRUE;
			_DFII_DBFetch.connectionIdent := _lConnectionIdent;
			_eStep := eSQLREQ_STEP_GETTIME_FETCH_r;

		eSQLREQ_STEP_GETTIME_FETCH_r:

			_DFII_DBFetch();

			IF _DFII_DBFetch.status = ERR_OK THEN

				_bCol := 1;
				_eStep := eSQLREQ_STEP_GETTIME_GETVAL;

			ELSIF _DFII_DBFetch.status <> ERR_FUB_BUSY THEN

				IF _DFII_DBFetch.dbError = DB_SQL_NO_DATA THEN

					_eStep := eSQLREQ_STEP_WAITFORCOMMAND;

				ELSE

					_sAction := 'Get Time failed (FETCH):';
					_eStep := eSQLREQ_STEP_GET_ERROR;

				END_IF

			END_IF

		(* Werte holen *)

		eSQLREQ_STEP_GETTIME_GETVAL:

			_DFII_GetData.enable := TRUE;
			_DFII_GetData.connectionIdent := _lConnectionIdent;
			_DFII_GetData.columnIdx := _bCol;

			_diTime := -1;
			_DFII_GetData.pData := ADR(_diTime);
			_DFII_GetData.dataSize := SIZEOF(_diTime);
			_DFII_GetData.dataType := DB_SQL_INTEGER;

			_eStep := eSQLREQ_STEP_GETTIME_GETVAL_r;

		eSQLREQ_STEP_GETTIME_GETVAL_r:

			_DFII_GetData();

			IF _DFII_GetData.status = ERR_OK THEN

				IF _diTime > 0 THEN

					_DTSetTime(enable := TRUE, DT1 := DINT_TO_DT(_diTime));

				END_IF

				_sLogEntryI := WSTRING_TO_STRING(IFmnParam.Out.utfMachineNumber);
				_sLogEntryI := CONCAT(_sLogEntryI, '-hlDFII$tSUCC$tGETTIME');
				_InsertRB(wPtrWrite := _wPtrRBwrite, wPtrRead := _wPtrRBread, wPtrStart := _wPtrRBstart);

				_eStep := eSQLREQ_STEP_WAITFORCOMMAND;

			ELSIF _DFII_GetData.status <> ERR_FUB_BUSY THEN
				_sAction := 'Get Time failed (VAL):';
				_eStep := eSQLREQ_STEP_GET_ERROR;
			END_IF

		(* Lese Fehler aus *)
		eSQLREQ_STEP_GET_ERROR:

			IF _lConnectionIdent = 0 THEN
				hlDFIIStat.sStatus := 'Connect failed !';
				_eStep := eSQLREQ_STEP_ERROR;
			ELSE
				brsmemset(ADR(hlDFIIStat.sStatus),0,SIZEOF(hlDFIIStat.sStatus));
				_DFII_DBErrMsg.enable := TRUE;
				_DFII_DBErrMsg.connectionIdent := _lConnectionIdent;
				_DFII_DBErrMsg.pErrorMessage := ADR(hlDFIIStat.sStatus);
				_DFII_DBErrMsg.errorMessageSize := SIZEOF(hlDFIIStat.sStatus);
				_eStep := eSQLREQ_STEP_GET_ERROR_r;
			END_IF

		(* Warte bis Fehler ausgelesen *)
		eSQLREQ_STEP_GET_ERROR_r:

			_DFII_DBErrMsg();

			IF _DFII_DBErrMsg.status = ERR_OK THEN

				_sLogEntryI := WSTRING_TO_STRING(IFmnParam.Out.utfMachineNumber);
				_sLogEntryI := CONCAT(_sLogEntryI, '-hlDFII$tWARN$t');
				_sLogEntryI := CONCAT(_sLogEntryI, _sAction);
				_sLogEntryI := CONCAT(_sLogEntryI, hlDFIIStat.sStatus);

				_eStep := eSQLREQ_STEP_LOGRB_ERROR;

			ELSIF _DFII_DBErrMsg.status <> ERR_FUB_BUSY THEN

				hlDFIIStat.sStatus := ' DBErrMsg.status = ';
				_sValue := UINT_TO_STRING(_DFII_DBErrMsg.status);
				hlDFIIStat.sStatus := CONCAT(hlDFIIStat.sStatus, _sValue);

				_sLogEntryI := WSTRING_TO_STRING(IFmnParam.Out.utfMachineNumber);
				_sLogEntryI := CONCAT(_sLogEntryI, '-hlDFII$tWARN$t');
				_sLogEntryI := CONCAT(_sLogEntryI, _sAction);
				_sLogEntryI := CONCAT(_sLogEntryI, hlDFIIStat.sStatus);

				_eStep := eSQLREQ_STEP_LOGRB_ERROR;

			END_IF

		eSQLREQ_STEP_LOGRB_ERROR:

			_InsertRB(wPtrWrite := _wPtrRBwrite, wPtrRead := _wPtrRBread, wPtrStart := _wPtrRBstart);
			_eStep := eSQLREQ_STEP_LOG_ERROR;

		eSQLREQ_STEP_LOG_ERROR:

			_kgArLogWrite.logLevel 	:= arlogLEVEL_WARNING;
			_kgArLogWrite.text		:= LEFT(_sLogEntryI, 127);
			_kgArLogWrite();

			IF _kgArLogWrite.status <> ERR_FUB_BUSY THEN
				brsmemset(ADR(_sLogEntryI), 0, SIZEOF(_sLogEntryI));
				_eStep := eSQLREQ_STEP_LOG_ERROR1;
			END_IF

		eSQLREQ_STEP_LOG_ERROR1:

			_kgArLogWrite.logLevel 	:= arlogLEVEL_WARNING;
			_kgArLogWrite.text		:= LEFT(_sSQLstring, 127);
			_kgArLogWrite();

			IF _kgArLogWrite.status <> ERR_FUB_BUSY THEN
				_eStep := eSQLREQ_STEP_ERROR;
			END_IF

		(* Fehlerschritt *)
		eSQLREQ_STEP_ERROR:

	END_CASE

END_ACTION
```

#### _CreateConnectionString.st - Connectionstring for SQL-Client
```iecst
(********************************************************************
 * COPYRIGHT -- Herbert Kannegiesser GmbH
 ********************************************************************
 * Program: hlDFII
 * File: _CreateConnectionString.st
 * Author: hunholz
 * Created: June 19, 2012
 ********************************************************************
 * Implementation of program hlDFII
 ********************************************************************)

(* Connectionstring for SQL-Client *)
FUNCTION_BLOCK _CreateConnectionString

	ConnString := USINT_TO_STRING(IP.bNetId1);
	ConnString := CONCAT(ConnString,'.');
	_sOkt := USINT_TO_STRING(IP.bNetId2);
	ConnString := CONCAT(ConnString,_sOkt);
	ConnString := CONCAT(ConnString,'.');
	_sOkt := USINT_TO_STRING(IP.bNetId3+Conn.bDBservReg);
	ConnString := CONCAT(ConnString,_sOkt);
	ConnString := CONCAT(ConnString,'.');
	_sOkt := USINT_TO_STRING(Conn.bDBservAdr);
	ConnString := CONCAT(ConnString,_sOkt);

	HostString := ConnString;

	_sInstance := Conn.sServInst;

	IF Conn.wDBservPort <> 0 THEN

		// Wenn der Port <> 0 ist, wird der SQL-Server direkt über den Port angesprochen

		ConnString := CONCAT(ConnString, ':');
		_sPort 	 := UINT_TO_STRING(Conn.wDBservPort);
		ConnString := CONCAT(ConnString, _sPort);

	ELSE

		// Wenn mit der Instanz gearbeitet wird, muss auf dem PC der SQL-Browser-Dienst laufen

		IF LEN(_sInstance) > 0 THEN

			REPEAT

				_iFound := FIND(_sInstance,' ');

				IF _iFound <> 0 THEN
					_sInstance := DELETE(_sInstance,1,_iFound);
				END_IF

				UNTIL
				_iFound = 0 OR LEN(_sInstance) = 0
			END_REPEAT

			IF LEN(_sInstance) > 0 THEN
				ConnString := CONCAT(ConnString, '\');
				ConnString := CONCAT(ConnString, _sInstance);
			END_IF

		END_IF

	END_IF

END_FUNCTION_BLOCK
```

#### hlDFII.fun
```iecst
(********************************************************************
 * COPYRIGHT -- Herbert Kannegiesser GmbH
 ********************************************************************
 * Program: hlDFII
 * File: hlDFII.fun
 * Author: hunholz
 * Created: June 19, 2012
 ********************************************************************
 * Functions and function blocks of program hlDFII
 ********************************************************************)

FUNCTION_BLOCK _CreateConnectionString (*Connectionstring for SQL-Client*)
	VAR_INPUT
		IP : mnEthIP_typ;
		Conn : hlDFIIParMacConn_typ;
	END_VAR
	VAR_OUTPUT
		ConnString : STRING[39];
		HostString : STRING[15];
	END_VAR
	VAR
		_sOkt : STRING[3];
		_sInstance : STRING[15];
		_sPort : STRING[5];
		_iFound : INT;
	END_VAR
END_FUNCTION_BLOCK
```

### hlDFII_History.txt
```
1.03.0		28.9.2011	AH Auf mnParam 0.05.0 umgestellt
1.04.0		11.10.2011	AH Auf mnParam 0.06.0 umgestellt, Maschinennummer kommt aus Datei
1.04.1		18.11.2011	AH Zwischenversion. Maschinenregistrierung startet jetzt automatisch.
						AH Attribute werden mit in die Meldungshistorie eingetragen
1.05.0		03.11.2011	AH Umstellung auf AS 3.0.90. IF ist eindeutig mit Ein- und Ausgangskanal definiert
			14.11.2011	AH Schnittstelle zu mnCnt umgestellt
1.06.0		21.12.2011	AH SPS-Log und UDP-Logging eingeführt
						AH Fehlerhandling geändert. Bei Fehlern wird grundsätzlich die Verbindung abgebaut.
1.07.0		03.01.2012	AH Packetversion wird in hlDFIIStatAd ausgegeben
1.08.0		12.01.2012	AH Kategorie-Programm-Zuordnung wird gecachet
1.09.0		24.01.2012	AH Anpassung an KGStandard 1.13.0 (Ringbuffer)
1.10.0		26.01.2012  AH Erweiterter Substatus für Zeitzähler mnCnt 0.14.0
1.10.1		07.02.2012  AH Schließendes Anführungszeichen im SQL-String Batch-Event für die MachineID fehlte
						AH Logeintrag erweitert
1.10.2		07.02.2012	AH Bei Batchevent mit 0 Teilposten hat sich die Sendeschrittkette aufgehängt
1.10.3		07.02.2012	AH GO ist kein gültiger TSQL-Befehl
1.10.4		07.02.2012	AH SQL-String Batchevent zu Debugzwecken kopiert. Log-String auf 511 Zeichen verlängert.
1.10.5		09.02.2012	AH Ziel- und Quellnamen für Postenevent ergänzt.
1.10.6		10.02.2012	AH Bei spInsEventStatItem_StateTime ein Komma zu viel
1.11.0		10.02.2012	AH Batchevent gibt jetzt immer Quell- und Zielort an. Dazu ist auch mnCnt 0.15.0 notwendig
1.11.1		10.02.2012	AH Wieder ein Komma zu viel
1.11.2		10.02.2012	AH Anführungszeichen hinter Maschinennummer oftmals zu wenig
1.11.3		10.02.2012	AH FromOutside und ToOutside müssen beim BatchEvent immer beide definiert sein
1.12.0		13.02.2012	AH Einige Korrekturen auf Anregung von Thomas Horn (Fehler in Strings, Komma usw.)
						   Anpassung an mnCnt 0.16.0
1.12.1		14.02.2012	AH Error-Logging erweitert und Debugging korrigiert. Logging-Port ist jetzt per Konstante definiert
						   HLDFII_UDP_PORT_LOG4NET
1.12.2		14.02.2012	AH Jetzt sollte auch der richtige String an Log4Net geschickt werden
1.13.0		20.02.2012	AH Client muss per Konfiguration freigeschaltet werden und kann per Parameter deaktiviert werden
							- Package gibt im IFhlDFII.Out.wStatus den aktuellen Status OK, Init oder Disabled aus (siehe Konstanten)
1.14.0		13.03.2012	AH Client muss per Konstante freigeschaltet werden. Andernfalls läuft er nicht an. Parameter von 1.13.0 entfallen wieder.
						   Mehr UDP-Logging
1.14.1		20.03.2012	AH Abhängigkeiten
1.14.2		28.03.2012	AH Bugfix: Logger. Parameter Start wurde nicht übergeben.
						   Connectionstring: Entweder Port oder Instanz.
1.15.0		03.04.2012	AH Category Cache entfernt.
						   xConnected eingeführt
1.16.0		11.04.2012	AH Maschinenregistrierung sendet jetzt auch den Maschinennamen
1.17.0		22.06.2012	AH Zweiter SQL-Client implementiert, der Maschinenstati und Postenverfolgungsinformationen meldet.
						   Kann unabhängig von DFII laufen.
						   ACHTUNG: Parameterstruktur hat sich verändert!!!
```

### Package Logical/Standard/Kanlink/KGFramework/Pkg_mnTest - Testadapter für automatische Tests

### Pkg_mnTest.typ - Package data types
```iecst
(********************************************************************
 * COPYRIGHT -- Herbert Kannegiesser GmbH
 ********************************************************************
 * Package: Pkg_mnTest
 * File: Pkg_mnTest.typ
 * Author: hunholz
 * Created: March 06, 2012
 ********************************************************************
 * Data types of package Pkg_mnTest
 ********************************************************************)

TYPE
	IFmnTestOut_typ : 	STRUCT
		xNoMessages : BOOL := FALSE;
	END_STRUCT;
	IFmnTestIn_typ : 	STRUCT
		pStrucTest : UDINT;
	END_STRUCT;
	IFmnTest_typ : 	STRUCT
		In : IFmnTestIn_typ;
		Out : IFmnTestOut_typ;
	END_STRUCT;
	mnTestStatAd_typ : 	STRUCT
		wMode : UINT; (*0 - deaktiviert. 1.. Nummer des Testmode*)
		sPkgVersion : STRING[10];
	END_STRUCT;
END_TYPE
```

### Pkg_mnTest.var - Package variables
```iecst
(********************************************************************
 * COPYRIGHT -- Herbert Kannegiesser GmbH
 ********************************************************************
 * Package: Pkg_mnTest
 * File: Pkg_mnTest.var
 * Author: hunholz
 * Created: March 06, 2012
 ********************************************************************
 * Variables of package Pkg_mnTest
 ********************************************************************)
VAR
	IFmnTest : IFmnTest_typ;
	mnTestCmd : KG_Cmd_typ;
	mnTestStatAd : mnTestStatAd_typ;
	mnTestStat : Stat_typ;
END_VAR
(*KONSTANTEN*)
VAR CONSTANT
	MNTEST_CMD_SETMODE : UINT := 1000; (*Mode steht in lData0*)
	MNTEST_CMD_RESET : UINT := 1001; (*Warm- oder Kaltstart, siehe lData0*)
	MNTEST_CMDSTAT_SETMODEFAILED : UINT := 60000;
	MNTEST_TESTMODE_INTERFACE : UINT := 1; (*Reiner Interfacetest*)
	MNTEST_TESTMODE_MAX : UINT := 2;
	MNTEST_RESETMODE_WARMSTART : USINT := 1;
	MNTEST_RESETMODE_COLDSTART : USINT := 2;
	MNTEST_STAT_ERRFBSETMODE : UINT := 60000; (*Fehler aus _fbSetMode. Siehe sStatus*)
	MNTEST_STAT_ERRMSGCFGCNT : UINT := 60001; (*Falsche Anzahl Meldungen*)
	MNTEST_STAT_ERRMSGCFG : UINT := 60002; (*Fehler DatObjInfo*)
	MNTEST_STAT_FBRUNTEST : UINT := 60003; (*Fehler aus _fbRunTest. Siehe sStatus*)
END_VAR
```

### Program Logical/Standard/Kanlink/KGFramework/Pkg_mnTest/mnTest (IEC) - Testadapter
